    |   movel([0.140704, -1.403542, -2.555417, -0.753429, 1.570796, 1.711500],accel_mss,speed_ms,0,blend_radius_m)
    |   movel([0.140545, -1.403137, -2.555717, -0.753535, 1.570796, 1.711342],accel_mss,speed_ms,0,blend_radius_m)
    |   movel([0.140518, -1.402670, -2.556062, -0.753657, 1.570796, 1.711315],accel_mss,speed_ms,0,blend_radius_m)
    |   movel([0.140843, -1.401367, -2.557021, -0.754000, 1.570796, 1.711640],accel_mss,speed_ms,0,blend_radius_m)
    |   movel([0.141778, -1.399330, -2.558517, -0.754541, 1.570796, 1.712574],accel_mss,speed_ms,0,blend_radius_m)
    |   movel([0.143948, -1.395292, -2.561465, -0.755632, 1.570796, 1.714744],accel_mss,speed_ms,0,blend_radius_m)
    |   movel([0.146129, -1.391761, -2.564023, -0.756605, 1.570796, 1.716925],accel_mss,speed_ms,0,blend_radius_m)
    |   movel([0.148288, -1.388770, -2.566175, -0.757443, 1.570796, 1.719084],accel_mss,speed_ms,0,blend_radius_m)
    |   movel([0.149299, -1.387556, -2.567045, -0.757787, 1.570796, 1.720095],accel_mss,speed_ms,0,blend_radius_m)
    |   movel([0.150400, -1.386385, -2.567883, -0.758121, 1.570796, 1.721196],accel_mss,speed_ms,0,blend_radius_m)
    |   movel([0.151006, -1.385809, -2.568294, -0.758286, 1.570796, 1.721802],accel_mss,speed_ms,0,blend_radius_m)
    |   movel([0.153931, -1.383309, -2.570072, -0.759008, 1.570796, 1.724727],accel_mss,speed_ms,0,blend_radius_m)
    |   movel([0.156335, -1.381241, -2.571537, -0.759611, 1.570796, 1.727131],accel_mss,speed_ms,0,blend_radius_m)
    |   movel([0.159846, -1.377963, -2.573845, -0.760581, 1.570796, 1.730642],accel_mss,speed_ms,0,blend_radius_m)
    |   movel([0.163498, -1.374419, -2.576324, -0.761646, 1.570796, 1.734295],accel_mss,speed_ms,0,blend_radius_m)
    |   movel([0.166495, -1.371353, -2.578454, -0.762582, 1.570796, 1.737291],accel_mss,speed_ms,0,blend_radius_m)
    |   movel([0.170128, -1.367386, -2.581189, -0.763813, 1.570796, 1.740924],accel_mss,speed_ms,0,blend_radius_m)
    |   movel([0.173632, -1.363310, -2.583978, -0.765102, 1.570796, 1.744429],accel_mss,speed_ms,0,blend_radius_m)
    |   movel([0.176951, -1.359183, -2.586776, -0.766430, 1.570796, 1.747747],accel_mss,speed_ms,0,blend_radius_m)
    |   movel([0.180116, -1.354961, -2.589615, -0.767813, 1.570796, 1.750913],accel_mss,speed_ms,0,blend_radius_m)
    |   movel([0.183146, -1.350616, -2.592510, -0.769263, 1.570796, 1.753942],accel_mss,speed_ms,0,blend_radius_m)
    |   movel([0.186004, -1.346192, -2.595432, -0.770766, 1.570796, 1.756800],accel_mss,speed_ms,0,blend_radius_m)
    |   movel([0.188766, -1.341570, -2.598454, -0.772364, 1.570796, 1.759562],accel_mss,speed_ms,0,blend_radius_m)
    |   movel([0.191358, -1.336888, -2.601487, -0.774014, 1.570796, 1.762154],accel_mss,speed_ms,0,blend_radius_m)
    |   movel([0.194463, -1.330702, -2.605447, -0.776239, 1.570796, 1.765259],accel_mss,speed_ms,0,blend_radius_m)
    |   movel([0.197247, -1.324446, -2.609400, -0.778543, 1.570796, 1.768044],accel_mss,speed_ms,0,blend_radius_m)
    |   movel([0.199689, -1.318160, -2.613319, -0.780910, 1.570796, 1.770485],accel_mss,speed_ms,0,blend_radius_m)
    |   movel([0.201775, -1.311845, -2.617204, -0.783340, 1.570796, 1.772572],accel_mss,speed_ms,0,blend_radius_m)
    |   movel([0.203479, -1.305580, -2.621005, -0.785804, 1.570796, 1.774275],accel_mss,speed_ms,0,blend_radius_m)
    |   movel([0.204799, -1.299337, -2.624742, -0.788310, 1.570796, 1.775595],accel_mss,speed_ms,0,blend_radius_m)
    |   movel([0.205703, -1.293227, -2.628351, -0.790810, 1.570796, 1.776499],accel_mss,speed_ms,0,blend_radius_m)
    |   movel([0.206187, -1.287198, -2.631865, -0.793325, 1.570796, 1.776984],accel_mss,speed_ms,0,blend_radius_m)
    |   movel([0.206497, -1.284112, -2.633647, -0.794631, 1.570796, 1.777293],accel_mss,speed_ms,0,blend_radius_m)
    |   movel([0.207150, -1.281572, -2.635103, -0.795714, 1.570796, 1.777946],accel_mss,speed_ms,0,blend_radius_m)
    |   movel([0.207592, -1.280512, -2.635709, -0.796168, 1.570796, 1.778388],accel_mss,speed_ms,0,blend_radius_m)
    |   movel([0.208169, -1.279450, -2.636314, -0.796625, 1.570796, 1.778966],accel_mss,speed_ms,0,blend_radius_m)
    |   movel([0.208820, -1.278512, -2.636847, -0.797030, 1.570796, 1.779616],accel_mss,speed_ms,0,blend_radius_m)
    |   movel([0.210185, -1.277059, -2.637671, -0.797659, 1.570796, 1.780981],accel_mss,speed_ms,0,blend_radius_m)
    |   movel([0.210558, -1.276782, -2.637828, -0.797779, 1.570796, 1.781354],accel_mss,speed_ms,0,blend_radius_m)
    |   movel([0.211690, -1.276412, -2.638038, -0.797940, 1.570796, 1.782486],accel_mss,speed_ms,0,blend_radius_m)
    |   movel([0.212752, -1.276292, -2.638105, -0.797992, 1.570796, 1.783548],accel_mss,speed_ms,0,blend_radius_m)
    |   movel([0.213684, -1.276450, -2.638016, -0.797923, 1.570796, 1.784480],accel_mss,speed_ms,0,blend_radius_m)
    |   movel([0.214653, -1.276937, -2.637741, -0.797712, 1.570796, 1.785449],accel_mss,speed_ms,0,blend_radius_m)
    |   movel([0.215875, -1.277874, -2.637209, -0.797305, 1.570796, 1.786671],accel_mss,speed_ms,0,blend_radius_m)
    |   movel([0.217446, -1.279458, -2.636309, -0.796622, 1.570796, 1.788242],accel_mss,speed_ms,0,blend_radius_m)
    |   movel([0.218701, -1.281264, -2.635279, -0.795846, 1.570796, 1.789497],accel_mss,speed_ms,0,blend_radius_m)
    |   movel([0.219663, -1.283334, -2.634093, -0.794961, 1.570796, 1.790460],accel_mss,speed_ms,0,blend_radius_m)
    |   movel([0.220360, -1.285698, -2.632733, -0.793959, 1.570796, 1.791157],accel_mss,speed_ms,0,blend_radius_m)
    |   movel([0.220698, -1.287639, -2.631610, -0.793140, 1.570796, 1.791494],accel_mss,speed_ms,0,blend_radius_m)
    |   movel([0.220907, -1.289828, -2.630338, -0.792223, 1.570796, 1.791703],accel_mss,speed_ms,0,blend_radius_m)
    |   movel([0.221010, -1.292587, -2.628727, -0.791076, 1.570796, 1.791806],accel_mss,speed_ms,0,blend_radius_m)
    |   movel([0.221047, -1.301875, -2.623229, -0.787285, 1.570796, 1.791843],accel_mss,speed_ms,0,blend_radius_m)
    |   movel([0.221214, -1.305714, -2.620925, -0.785751, 1.570796, 1.792010],accel_mss,speed_ms,0,blend_radius_m)
    |   movel([0.221547, -1.308582, -2.619190, -0.784617, 1.570796, 1.792343],accel_mss,speed_ms,0,blend_radius_m)
    |   movel([0.222085, -1.310928, -2.617763, -0.783698, 1.570796, 1.792881],accel_mss,speed_ms,0,blend_radius_m)
    |   movel([0.223013, -1.312969, -2.616516, -0.782904, 1.570796, 1.793809],accel_mss,speed_ms,0,blend_radius_m)
    |   movel([0.223526, -1.313486, -2.616199, -0.782704, 1.570796, 1.794322],accel_mss,speed_ms,0,blend_radius_m)
    |   movel([0.224254, -1.313767, -2.616027, -0.782595, 1.570796, 1.795050],accel_mss,speed_ms,0,blend_radius_m)
    |   movel([0.225101, -1.313780, -2.616019, -0.782590, 1.570796, 1.795897],accel_mss,speed_ms,0,blend_radius_m)
    |   movel([0.226034, -1.313522, -2.616177, -0.782690, 1.570796, 1.796830],accel_mss,speed_ms,0,blend_radius_m)
    |   movel([0.227364, -1.312916, -2.616548, -0.782924, 1.570796, 1.798160],accel_mss,speed_ms,0,blend_radius_m)
    |   movel([0.228675, -1.312190, -2.616993, -0.783206, 1.570796, 1.799471],accel_mss,speed_ms,0,blend_radius_m)
    |   movel([0.230649, -1.310918, -2.617770, -0.783702, 1.570796, 1.801445],accel_mss,speed_ms,0,blend_radius_m)
    |   movel([0.232595, -1.309499, -2.618633, -0.784257, 1.570796, 1.803392],accel_mss,speed_ms,0,blend_radius_m)
    |   movel([0.234895, -1.307655, -2.619752, -0.784982, 1.570796, 1.805692],accel_mss,speed_ms,0,blend_radius_m)
    |   movel([0.241204, -1.302298, -2.622976, -0.787115, 1.570796, 1.812000],accel_mss,speed_ms,0,blend_radius_m)
    |   movel([0.243555, -1.300425, -2.624095, -0.787869, 1.570796, 1.814351],accel_mss,speed_ms,0,blend_radius_m)
    |   movel([0.245404, -1.299103, -2.624882, -0.788405, 1.570796, 1.816201],accel_mss,speed_ms,0,blend_radius_m)
    |   movel([0.246945, -1.298199, -2.625419, -0.788772, 1.570796, 1.817741],accel_mss,speed_ms,0,blend_radius_m)
    |   movel([0.247792, -1.297825, -2.625640, -0.788924, 1.570796, 1.818588],accel_mss,speed_ms,0,blend_radius_m)
    |   movel([0.248634, -1.297559, -2.625797, -0.789032, 1.570796, 1.819430],accel_mss,speed_ms,0,blend_radius_m)
    |   movel([0.249248, -1.297496, -2.625835, -0.789058, 1.570796, 1.820044],accel_mss,speed_ms,0,blend_radius_m)
    |   movel([0.249761, -1.297629, -2.625756, -0.789004, 1.570796, 1.820557],accel_mss,speed_ms,0,blend_radius_m)
    |   movel([0.250158, -1.297955, -2.625563, -0.788871, 1.570796, 1.820954],accel_mss,speed_ms,0,blend_radius_m)
    |   movel([0.250380, -1.298428, -2.625282, -0.788679, 1.570796, 1.821176],accel_mss,speed_ms,0,blend_radius_m)
    |   movel([0.250519, -1.300019, -2.624337, -0.788033, 1.570796, 1.821316],accel_mss,speed_ms,0,blend_radius_m)
    |   movel([0.250460, -1.300588, -2.623997, -0.787803, 1.570796, 1.821256],accel_mss,speed_ms,0,blend_radius_m)
    |   movel([0.250051, -1.302510, -2.622849, -0.787030, 1.570796, 1.820848],accel_mss,speed_ms,0,blend_radius_m)
    |   speed_ms = 0.005
    |   movel([0.250051, -1.293311, -2.618501, -0.800577, 1.570796, 1.820848],accel_mss,speed_ms,0,blend_radius_m)
    |   speed_ms = 0.040
    |   movel([0.285051, -1.248291, -2.643835, -0.820263, 1.570796, 1.855847],accel_mss,speed_ms,0,blend_radius_m)
    |   speed_ms = 0.005
    |   movel([0.285051, -1.257727, -2.648387, -0.806275, 1.570796, 1.855847],accel_mss,speed_ms,0,blend_radius_m)
    |   speed_ms = 0.025
    |   movel([0.285376, -1.257416, -2.648555, -0.806417, 1.570796, 1.856173],accel_mss,speed_ms,0,blend_radius_m)
    |   movel([0.285614, -1.256958, -2.648804, -0.806628, 1.570796, 1.856410],accel_mss,speed_ms,0,blend_radius_m)
    |   movel([0.285837, -1.256166, -2.649232, -0.806991, 1.570796, 1.856634],accel_mss,speed_ms,0,blend_radius_m)
    |   movel([0.286186, -1.254460, -2.650153, -0.807777, 1.570796, 1.856982],accel_mss,speed_ms,0,blend_radius_m)
    |   movel([0.286743, -1.250478, -2.652287, -0.809624, 1.570796, 1.857539],accel_mss,speed_ms,0,blend_radius_m)
    |   movel([0.286878, -1.248468, -2.653357, -0.810563, 1.570796, 1.857674],accel_mss,speed_ms,0,blend_radius_m)
    |   movel([0.286872, -1.244744, -2.655328, -0.812317, 1.570796, 1.857668],accel_mss,speed_ms,0,blend_radius_m)
    |   movel([0.286986, -1.244540, -2.655435, -0.812414, 1.570796, 1.857783],accel_mss,speed_ms,0,blend_radius_m)
    |   movel([0.287202, -1.244420, -2.655498, -0.812470, 1.570796, 1.857998],accel_mss,speed_ms,0,blend_radius_m)
    |   movel([0.287547, -1.244241, -2.655593, -0.812555, 1.570796, 1.858343],accel_mss,speed_ms,0,blend_radius_m)
    |   movel([0.287781, -1.243914, -2.655765, -0.812710, 1.570796, 1.858577],accel_mss,speed_ms,0,blend_radius_m)
    |   movel([0.288488, -1.241734, -2.656909, -0.813747, 1.570796, 1.859284],accel_mss,speed_ms,0,blend_radius_m)
    |   movel([0.289030, -1.239404, -2.658125, -0.814861, 1.570796, 1.859827],accel_mss,speed_ms,0,blend_radius_m)
    |   movel([0.289144, -1.237626, -2.659048, -0.815715, 1.570796, 1.859940],accel_mss,speed_ms,0,blend_radius_m)
    |   movel([0.289053, -1.236830, -2.659460, -0.816098, 1.570796, 1.859850],accel_mss,speed_ms,0,blend_radius_m)
    |   movel([0.288864, -1.236454, -2.659655, -0.816280, 1.570796, 1.859660],accel_mss,speed_ms,0,blend_radius_m)
    |   movel([0.288563, -1.236423, -2.659671, -0.816295, 1.570796, 1.859359],accel_mss,speed_ms,0,blend_radius_m)
    |   movel([0.288157, -1.236673, -2.659542, -0.816174, 1.570796, 1.858953],accel_mss,speed_ms,0,blend_radius_m)
    |   movel([0.287954, -1.236902, -2.659423, -0.816064, 1.570796, 1.858750],accel_mss,speed_ms,0,blend_radius_m)
    |   movel([0.287849, -1.237125, -2.659308, -0.815956, 1.570796, 1.858646],accel_mss,speed_ms,0,blend_radius_m)
    |   movel([0.287893, -1.238385, -2.658654, -0.815350, 1.570796, 1.858690],accel_mss,speed_ms,0,blend_radius_m)
    |   movel([0.287887, -1.238901, -2.658386, -0.815102, 1.570796, 1.858683],accel_mss,speed_ms,0,blend_radius_m)
    |   movel([0.287513, -1.241756, -2.656897, -0.813736, 1.570796, 1.858309],accel_mss,speed_ms,0,blend_radius_m)
    |   movel([0.286745, -1.241225, -2.657175, -0.813990, 1.570796, 1.857541],accel_mss,speed_ms,0,blend_radius_m)
    |   movel([0.285897, -1.240581, -2.657511, -0.814297, 1.570796, 1.856693],accel_mss,speed_ms,0,blend_radius_m)
    |   movel([0.285614, -1.240567, -2.657518, -0.814304, 1.570796, 1.856410],accel_mss,speed_ms,0,blend_radius_m)
    |   movel([0.285291, -1.240759, -2.657418, -0.814212, 1.570796, 1.856087],accel_mss,speed_ms,0,blend_radius_m)
    |   movel([0.285032, -1.241098, -2.657241, -0.814050, 1.570796, 1.855828],accel_mss,speed_ms,0,blend_radius_m)
    |   movel([0.284949, -1.241441, -2.657062, -0.813886, 1.570796, 1.855745],accel_mss,speed_ms,0,blend_radius_m)
    |   movel([0.285127, -1.242733, -2.656385, -0.813271, 1.570796, 1.855923],accel_mss,speed_ms,0,blend_radius_m)
    |   movel([0.285518, -1.245087, -2.655147, -0.812155, 1.570796, 1.856314],accel_mss,speed_ms,0,blend_radius_m)
    |   movel([0.285650, -1.247822, -2.653700, -0.810866, 1.570796, 1.856446],accel_mss,speed_ms,0,blend_radius_m)
    |   movel([0.285532, -1.250774, -2.652129, -0.809486, 1.570796, 1.856328],accel_mss,speed_ms,0,blend_radius_m)
    |   movel([0.285165, -1.253795, -2.650510, -0.808083, 1.570796, 1.855962],accel_mss,speed_ms,0,blend_radius_m)
    |   movel([0.285029, -1.254644, -2.650053, -0.807692, 1.570796, 1.855825],accel_mss,speed_ms,0,blend_radius_m)
    |   movel([0.284302, -1.253909, -2.650449, -0.808031, 1.570796, 1.855098],accel_mss,speed_ms,0,blend_radius_m)
    |   movel([0.283800, -1.253480, -2.650679, -0.808229, 1.570796, 1.854597],accel_mss,speed_ms,0,blend_radius_m)
    |   movel([0.283333, -1.253283, -2.650785, -0.808320, 1.570796, 1.854130],accel_mss,speed_ms,0,blend_radius_m)
    |   movel([0.282930, -1.253309, -2.650771, -0.808308, 1.570796, 1.853726],accel_mss,speed_ms,0,blend_radius_m)
    |   movel([0.282597, -1.253538, -2.650648, -0.808202, 1.570796, 1.853393],accel_mss,speed_ms,0,blend_radius_m)
    |   movel([0.282529, -1.253687, -2.650569, -0.808134, 1.570796, 1.853326],accel_mss,speed_ms,0,blend_radius_m)
    |   movel([0.282510, -1.258156, -2.648154, -0.806079, 1.570796, 1.853306],accel_mss,speed_ms,0,blend_radius_m)
    |   movel([0.282198, -1.261061, -2.646572, -0.804757, 1.570796, 1.852994],accel_mss,speed_ms,0,blend_radius_m)
    |   movel([0.281587, -1.264059, -2.644927, -0.803402, 1.570796, 1.852383],accel_mss,speed_ms,0,blend_radius_m)
    |   movel([0.280691, -1.267080, -2.643260, -0.802049, 1.570796, 1.851487],accel_mss,speed_ms,0,blend_radius_m)
    |   movel([0.279427, -1.270591, -2.641308, -0.800490, 1.570796, 1.850224],accel_mss,speed_ms,0,blend_radius_m)
    |   movel([0.278962, -1.271746, -2.640662, -0.799981, 1.570796, 1.849758],accel_mss,speed_ms,0,blend_radius_m)
    |   movel([0.278807, -1.271873, -2.640591, -0.799925, 1.570796, 1.849604],accel_mss,speed_ms,0,blend_radius_m)
    |   movel([0.277931, -1.270373, -2.641430, -0.800587, 1.570796, 1.848727],accel_mss,speed_ms,0,blend_radius_m)
    |   movel([0.277769, -1.270303, -2.641468, -0.800618, 1.570796, 1.848565],accel_mss,speed_ms,0,blend_radius_m)
    |   movel([0.277540, -1.270378, -2.641427, -0.800584, 1.570796, 1.848337],accel_mss,speed_ms,0,blend_radius_m)
    |   movel([0.277044, -1.270862, -2.641156, -0.800370, 1.570796, 1.847840],accel_mss,speed_ms,0,blend_radius_m)
    |   movel([0.276091, -1.272411, -2.640290, -0.799688, 1.570796, 1.846887],accel_mss,speed_ms,0,blend_radius_m)
    |   movel([0.274985, -1.274185, -2.639293, -0.798910, 1.570796, 1.845782],accel_mss,speed_ms,0,blend_radius_m)
    |   movel([0.272593, -1.277484, -2.637431, -0.797474, 1.570796, 1.843389],accel_mss,speed_ms,0,blend_radius_m)
    |   movel([0.271336, -1.278966, -2.636589, -0.796834, 1.570796, 1.842132],accel_mss,speed_ms,0,blend_radius_m)
    |   movel([0.268622, -1.281745, -2.635004, -0.795640, 1.570796, 1.839418],accel_mss,speed_ms,0,blend_radius_m)
    |   movel([0.267067, -1.283243, -2.634146, -0.795001, 1.570796, 1.837863],accel_mss,speed_ms,0,blend_radius_m)
    |   movel([0.266749, -1.283416, -2.634046, -0.794927, 1.570796, 1.837545],accel_mss,speed_ms,0,blend_radius_m)
    |   movel([0.267003, -1.282685, -2.634466, -0.795238, 1.570796, 1.837799],accel_mss,speed_ms,0,blend_radius_m)
    |   movel([0.267156, -1.282373, -2.634645, -0.795372, 1.570796, 1.837953],accel_mss,speed_ms,0,blend_radius_m)
    |   movel([0.267374, -1.281632, -2.635069, -0.795688, 1.570796, 1.838171],accel_mss,speed_ms,0,blend_radius_m)
    |   movel([0.267265, -1.281398, -2.635202, -0.795788, 1.570796, 1.838061],accel_mss,speed_ms,0,blend_radius_m)
    |   movel([0.267029, -1.281290, -2.635264, -0.795835, 1.570796, 1.837826],accel_mss,speed_ms,0,blend_radius_m)
    |   movel([0.266711, -1.281327, -2.635243, -0.795819, 1.570796, 1.837507],accel_mss,speed_ms,0,blend_radius_m)
    |   movel([0.266379, -1.281504, -2.635142, -0.795743, 1.570796, 1.837175],accel_mss,speed_ms,0,blend_radius_m)
    |   movel([0.264753, -1.282545, -2.634546, -0.795298, 1.570796, 1.835550],accel_mss,speed_ms,0,blend_radius_m)
    |   movel([0.262799, -1.283498, -2.633999, -0.794892, 1.570796, 1.833595],accel_mss,speed_ms,0,blend_radius_m)
    |   movel([0.260794, -1.284240, -2.633572, -0.794576, 1.570796, 1.831590],accel_mss,speed_ms,0,blend_radius_m)
    |   movel([0.259009, -1.284664, -2.633329, -0.794397, 1.570796, 1.829805],accel_mss,speed_ms,0,blend_radius_m)
    |   movel([0.257566, -1.284887, -2.633200, -0.794302, 1.570796, 1.828363],accel_mss,speed_ms,0,blend_radius_m)
    |   movel([0.258580, -1.284223, -2.633582, -0.794583, 1.570796, 1.829377],accel_mss,speed_ms,0,blend_radius_m)
    |   movel([0.260055, -1.283172, -2.634187, -0.795031, 1.570796, 1.830851],accel_mss,speed_ms,0,blend_radius_m)
    |   movel([0.260356, -1.282858, -2.634366, -0.795164, 1.570796, 1.831153],accel_mss,speed_ms,0,blend_radius_m)
    |   movel([0.260526, -1.282508, -2.634567, -0.795314, 1.570796, 1.831322],accel_mss,speed_ms,0,blend_radius_m)
    |   movel([0.260492, -1.282266, -2.634706, -0.795417, 1.570796, 1.831289],accel_mss,speed_ms,0,blend_radius_m)
    |   movel([0.260273, -1.282178, -2.634756, -0.795455, 1.570796, 1.831070],accel_mss,speed_ms,0,blend_radius_m)
    |   movel([0.257760, -1.282555, -2.634540, -0.795294, 1.570796, 1.828556],accel_mss,speed_ms,0,blend_radius_m)
    |   movel([0.257143, -1.282548, -2.634544, -0.795297, 1.570796, 1.827940],accel_mss,speed_ms,0,blend_radius_m)
    |   movel([0.255004, -1.282200, -2.634744, -0.795445, 1.570796, 1.825800],accel_mss,speed_ms,0,blend_radius_m)
    |   movel([0.253443, -1.281754, -2.634999, -0.795636, 1.570796, 1.824239],accel_mss,speed_ms,0,blend_radius_m)
    |   movel([0.250378, -1.280508, -2.635711, -0.796170, 1.570796, 1.821175],accel_mss,speed_ms,0,blend_radius_m)
    |   movel([0.248859, -1.279752, -2.636142, -0.796495, 1.570796, 1.819656],accel_mss,speed_ms,0,blend_radius_m)
    |   movel([0.250690, -1.278643, -2.636773, -0.796973, 1.570796, 1.821486],accel_mss,speed_ms,0,blend_radius_m)
    |   movel([0.251682, -1.278031, -2.637120, -0.797238, 1.570796, 1.822478],accel_mss,speed_ms,0,blend_radius_m)
    |   movel([0.252495, -1.277367, -2.637497, -0.797525, 1.570796, 1.823292],accel_mss,speed_ms,0,blend_radius_m)
    |   movel([0.252645, -1.277082, -2.637658, -0.797649, 1.570796, 1.823441],accel_mss,speed_ms,0,blend_radius_m)
    |   movel([0.252625, -1.276826, -2.637803, -0.797760, 1.570796, 1.823422],accel_mss,speed_ms,0,blend_radius_m)
    |   movel([0.252420, -1.276660, -2.637897, -0.797832, 1.570796, 1.823216],accel_mss,speed_ms,0,blend_radius_m)
    |   movel([0.250730, -1.276368, -2.638062, -0.797959, 1.570796, 1.821526],accel_mss,speed_ms,0,blend_radius_m)
    |   movel([0.248210, -1.275930, -2.638310, -0.798149, 1.570796, 1.819007],accel_mss,speed_ms,0,blend_radius_m)
    |   movel([0.245957, -1.275281, -2.638676, -0.798432, 1.570796, 1.816753],accel_mss,speed_ms,0,blend_radius_m)
    |   movel([0.243901, -1.274399, -2.639173, -0.798817, 1.570796, 1.814697],accel_mss,speed_ms,0,blend_radius_m)
    |   movel([0.241981, -1.273254, -2.639817, -0.799318, 1.570796, 1.812778],accel_mss,speed_ms,0,blend_radius_m)
    |   movel([0.240628, -1.272326, -2.640337, -0.799726, 1.570796, 1.811424],accel_mss,speed_ms,0,blend_radius_m)
    |   movel([0.242149, -1.271884, -2.640585, -0.799920, 1.570796, 1.812945],accel_mss,speed_ms,0,blend_radius_m)
    |   movel([0.243577, -1.271407, -2.640852, -0.800130, 1.570796, 1.814374],accel_mss,speed_ms,0,blend_radius_m)
    |   movel([0.244768, -1.270870, -2.641152, -0.800367, 1.570796, 1.815564],accel_mss,speed_ms,0,blend_radius_m)
    |   movel([0.245620, -1.270334, -2.641451, -0.800604, 1.570796, 1.816416],accel_mss,speed_ms,0,blend_radius_m)
    |   movel([0.245834, -1.270117, -2.641572, -0.800700, 1.570796, 1.816631],accel_mss,speed_ms,0,blend_radius_m)
    |   movel([0.245956, -1.269872, -2.641709, -0.800808, 1.570796, 1.816753],accel_mss,speed_ms,0,blend_radius_m)
    |   movel([0.245937, -1.269634, -2.641841, -0.800913, 1.570796, 1.816733],accel_mss,speed_ms,0,blend_radius_m)
    |   movel([0.245749, -1.269477, -2.641929, -0.800983, 1.570796, 1.816546],accel_mss,speed_ms,0,blend_radius_m)
    |   movel([0.244338, -1.269231, -2.642066, -0.801092, 1.570796, 1.815134],accel_mss,speed_ms,0,blend_radius_m)
    |   movel([0.243592, -1.269121, -2.642127, -0.801141, 1.570796, 1.814389],accel_mss,speed_ms,0,blend_radius_m)
    |   movel([0.241491, -1.268600, -2.642417, -0.801372, 1.570796, 1.812287],accel_mss,speed_ms,0,blend_radius_m)
    |   movel([0.240267, -1.268026, -2.642736, -0.801628, 1.570796, 1.811064],accel_mss,speed_ms,0,blend_radius_m)
    |   movel([0.237751, -1.266229, -2.643731, -0.802429, 1.570796, 1.808548],accel_mss,speed_ms,0,blend_radius_m)
    |   movel([0.236809, -1.265256, -2.644268, -0.802865, 1.570796, 1.807606],accel_mss,speed_ms,0,blend_radius_m)
    |   movel([0.234505, -1.262022, -2.646046, -0.804321, 1.570796, 1.805301],accel_mss,speed_ms,0,blend_radius_m)
    |   movel([0.233410, -1.260262, -2.647008, -0.805119, 1.570796, 1.804207],accel_mss,speed_ms,0,blend_radius_m)
    |   movel([0.233543, -1.260074, -2.647110, -0.805205, 1.570796, 1.804339],accel_mss,speed_ms,0,blend_radius_m)
    |   movel([0.234795, -1.260230, -2.647025, -0.805134, 1.570796, 1.805592],accel_mss,speed_ms,0,blend_radius_m)
    |   movel([0.235308, -1.260299, -2.646987, -0.805102, 1.570796, 1.806104],accel_mss,speed_ms,0,blend_radius_m)
    |   movel([0.237799, -1.260349, -2.646961, -0.805080, 1.570796, 1.808596],accel_mss,speed_ms,0,blend_radius_m)
    |   movel([0.238169, -1.260286, -2.646995, -0.805108, 1.570796, 1.808965],accel_mss,speed_ms,0,blend_radius_m)
    |   movel([0.238709, -1.259961, -2.647172, -0.805256, 1.570796, 1.809505],accel_mss,speed_ms,0,blend_radius_m)
    |   movel([0.238960, -1.259624, -2.647356, -0.805410, 1.570796, 1.809756],accel_mss,speed_ms,0,blend_radius_m)
    |   movel([0.238957, -1.259371, -2.647493, -0.805524, 1.570796, 1.809753],accel_mss,speed_ms,0,blend_radius_m)
    |   movel([0.238642, -1.259153, -2.647612, -0.805624, 1.570796, 1.809439],accel_mss,speed_ms,0,blend_radius_m)
    |   movel([0.236421, -1.258302, -2.648074, -0.806012, 1.570796, 1.807218],accel_mss,speed_ms,0,blend_radius_m)
    |   movel([0.235003, -1.257497, -2.648511, -0.806380, 1.570796, 1.805800],accel_mss,speed_ms,0,blend_radius_m)
    |   movel([0.233648, -1.256526, -2.649037, -0.806826, 1.570796, 1.804444],accel_mss,speed_ms,0,blend_radius_m)
    |   movel([0.232494, -1.255470, -2.649608, -0.807311, 1.570796, 1.803290],accel_mss,speed_ms,0,blend_radius_m)
    |   movel([0.230105, -1.252420, -2.651248, -0.808720, 1.570796, 1.800901],accel_mss,speed_ms,0,blend_radius_m)
    |   movel([0.228663, -1.250377, -2.652341, -0.809671, 1.570796, 1.799459],accel_mss,speed_ms,0,blend_radius_m)
    |   movel([0.228616, -1.250017, -2.652533, -0.809839, 1.570796, 1.799412],accel_mss,speed_ms,0,blend_radius_m)
    |   movel([0.229564, -1.250008, -2.652538, -0.809843, 1.570796, 1.800360],accel_mss,speed_ms,0,blend_radius_m)
    |   movel([0.229992, -1.250043, -2.652519, -0.809827, 1.570796, 1.800788],accel_mss,speed_ms,0,blend_radius_m)
    |   movel([0.231557, -1.249933, -2.652578, -0.809878, 1.570796, 1.802353],accel_mss,speed_ms,0,blend_radius_m)
    |   movel([0.232180, -1.249807, -2.652645, -0.809937, 1.570796, 1.802977],accel_mss,speed_ms,0,blend_radius_m)
    |   movel([0.232659, -1.249546, -2.652784, -0.810059, 1.570796, 1.803455],accel_mss,speed_ms,0,blend_radius_m)
    |   movel([0.232791, -1.249316, -2.652907, -0.810167, 1.570796, 1.803588],accel_mss,speed_ms,0,blend_radius_m)
    |   movel([0.232794, -1.249067, -2.653039, -0.810283, 1.570796, 1.803590],accel_mss,speed_ms,0,blend_radius_m)
    |   movel([0.232586, -1.248795, -2.653184, -0.810410, 1.570796, 1.803382],accel_mss,speed_ms,0,blend_radius_m)
    |   movel([0.231381, -1.247999, -2.653607, -0.810783, 1.570796, 1.802178],accel_mss,speed_ms,0,blend_radius_m)
    |   movel([0.229753, -1.246883, -2.654198, -0.811308, 1.570796, 1.800549],accel_mss,speed_ms,0,blend_radius_m)
    |   movel([0.227669, -1.245075, -2.655153, -0.812160, 1.570796, 1.798465],accel_mss,speed_ms,0,blend_radius_m)
    |   movel([0.225697, -1.243153, -2.656165, -0.813072, 1.570796, 1.796493],accel_mss,speed_ms,0,blend_radius_m)
    |   movel([0.224468, -1.241636, -2.656959, -0.813793, 1.570796, 1.795264],accel_mss,speed_ms,0,blend_radius_m)
    |   movel([0.224133, -1.241124, -2.657228, -0.814038, 1.570796, 1.794929],accel_mss,speed_ms,0,blend_radius_m)
    |   movel([0.223619, -1.240166, -2.657728, -0.814496, 1.570796, 1.794415],accel_mss,speed_ms,0,blend_radius_m)
    |   movel([0.226300, -1.239267, -2.658196, -0.814926, 1.570796, 1.797097],accel_mss,speed_ms,0,blend_radius_m)
    |   movel([0.226990, -1.238984, -2.658343, -0.815062, 1.570796, 1.797786],accel_mss,speed_ms,0,blend_radius_m)
    |   movel([0.227360, -1.238690, -2.658496, -0.815203, 1.570796, 1.798157],accel_mss,speed_ms,0,blend_radius_m)
    |   movel([0.227525, -1.238345, -2.658675, -0.815369, 1.570796, 1.798322],accel_mss,speed_ms,0,blend_radius_m)
    |   movel([0.227501, -1.238151, -2.658776, -0.815462, 1.570796, 1.798297],accel_mss,speed_ms,0,blend_radius_m)
    |   movel([0.227391, -1.238029, -2.658839, -0.815521, 1.570796, 1.798188],accel_mss,speed_ms,0,blend_radius_m)
    |   movel([0.225593, -1.237852, -2.658931, -0.815606, 1.570796, 1.796390],accel_mss,speed_ms,0,blend_radius_m)
    |   movel([0.223952, -1.237328, -2.659202, -0.815858, 1.570796, 1.794749],accel_mss,speed_ms,0,blend_radius_m)
    |   movel([0.218123, -1.234687, -2.660567, -0.817135, 1.570796, 1.788919],accel_mss,speed_ms,0,blend_radius_m)
    |   movel([0.216800, -1.234048, -2.660896, -0.817445, 1.570796, 1.787597],accel_mss,speed_ms,0,blend_radius_m)
    |   movel([0.220608, -1.232835, -2.661519, -0.818035, 1.570796, 1.791404],accel_mss,speed_ms,0,blend_radius_m)
    |   movel([0.220926, -1.232640, -2.661619, -0.818130, 1.570796, 1.791722],accel_mss,speed_ms,0,blend_radius_m)
    |   movel([0.221103, -1.232409, -2.661737, -0.818243, 1.570796, 1.791900],accel_mss,speed_ms,0,blend_radius_m)
    |   movel([0.221168, -1.232051, -2.661920, -0.818417, 1.570796, 1.791964],accel_mss,speed_ms,0,blend_radius_m)
    |   movel([0.221038, -1.231793, -2.662052, -0.818543, 1.570796, 1.791834],accel_mss,speed_ms,0,blend_radius_m)
    |   movel([0.220136, -1.231236, -2.662337, -0.818816, 1.570796, 1.790932],accel_mss,speed_ms,0,blend_radius_m)
    |   movel([0.218436, -1.230663, -2.662630, -0.819096, 1.570796, 1.789232],accel_mss,speed_ms,0,blend_radius_m)
    |   movel([0.215494, -1.229992, -2.662972, -0.819425, 1.570796, 1.786290],accel_mss,speed_ms,0,blend_radius_m)
    |   movel([0.211124, -1.229342, -2.663303, -0.819744, 1.570796, 1.781921],accel_mss,speed_ms,0,blend_radius_m)
    |   movel([0.209198, -1.229270, -2.663340, -0.819780, 1.570796, 1.779994],accel_mss,speed_ms,0,blend_radius_m)
    |   movel([0.207322, -1.229351, -2.663298, -0.819740, 1.570796, 1.778118],accel_mss,speed_ms,0,blend_radius_m)
    |   movel([0.205959, -1.229442, -2.663252, -0.819695, 1.570796, 1.776755],accel_mss,speed_ms,0,blend_radius_m)
    |   movel([0.205889, -1.229255, -2.663347, -0.819787, 1.570796, 1.776685],accel_mss,speed_ms,0,blend_radius_m)
    |   movel([0.206212, -1.228981, -2.663486, -0.819921, 1.570796, 1.777008],accel_mss,speed_ms,0,blend_radius_m)
    |   movel([0.207881, -1.228399, -2.663782, -0.820207, 1.570796, 1.778677],accel_mss,speed_ms,0,blend_radius_m)
    |   movel([0.208910, -1.228042, -2.663964, -0.820384, 1.570796, 1.779707],accel_mss,speed_ms,0,blend_radius_m)
    |   movel([0.209651, -1.227627, -2.664174, -0.820588, 1.570796, 1.780447],accel_mss,speed_ms,0,blend_radius_m)
    |   movel([0.209813, -1.227371, -2.664304, -0.820714, 1.570796, 1.780610],accel_mss,speed_ms,0,blend_radius_m)
    |   movel([0.209810, -1.227135, -2.664423, -0.820831, 1.570796, 1.780606],accel_mss,speed_ms,0,blend_radius_m)
    |   movel([0.209627, -1.226934, -2.664525, -0.820930, 1.570796, 1.780424],accel_mss,speed_ms,0,blend_radius_m)
    |   movel([0.208422, -1.226483, -2.664753, -0.821153, 1.570796, 1.779219],accel_mss,speed_ms,0,blend_radius_m)
    |   movel([0.205590, -1.225749, -2.665124, -0.821516, 1.570796, 1.776387],accel_mss,speed_ms,0,blend_radius_m)
    |   movel([0.202937, -1.225278, -2.665361, -0.821749, 1.570796, 1.773733],accel_mss,speed_ms,0,blend_radius_m)
    |   movel([0.200496, -1.225073, -2.665465, -0.821852, 1.570796, 1.771292],accel_mss,speed_ms,0,blend_radius_m)
    |   movel([0.198313, -1.225138, -2.665432, -0.821819, 1.570796, 1.769109],accel_mss,speed_ms,0,blend_radius_m)
    |   movel([0.196815, -1.225270, -2.665365, -0.821754, 1.570796, 1.767612],accel_mss,speed_ms,0,blend_radius_m)
    |   movel([0.196665, -1.225161, -2.665420, -0.821808, 1.570796, 1.767461],accel_mss,speed_ms,0,blend_radius_m)
    |   movel([0.196789, -1.224942, -2.665530, -0.821916, 1.570796, 1.767585],accel_mss,speed_ms,0,blend_radius_m)
    |   movel([0.198166, -1.223979, -2.666015, -0.822395, 1.570796, 1.768963],accel_mss,speed_ms,0,blend_radius_m)
    |   movel([0.198894, -1.223467, -2.666272, -0.822649, 1.570796, 1.769690],accel_mss,speed_ms,0,blend_radius_m)
    |   movel([0.200219, -1.222435, -2.666790, -0.823164, 1.570796, 1.771015],accel_mss,speed_ms,0,blend_radius_m)
    |   movel([0.200325, -1.222080, -2.666968, -0.823342, 1.570796, 1.771122],accel_mss,speed_ms,0,blend_radius_m)
    |   movel([0.200128, -1.221809, -2.667103, -0.823477, 1.570796, 1.770925],accel_mss,speed_ms,0,blend_radius_m)
    |   movel([0.199567, -1.221632, -2.667191, -0.823565, 1.570796, 1.770363],accel_mss,speed_ms,0,blend_radius_m)
    |   movel([0.198593, -1.221552, -2.667232, -0.823605, 1.570796, 1.769390],accel_mss,speed_ms,0,blend_radius_m)
    |   movel([0.196633, -1.221578, -2.667219, -0.823592, 1.570796, 1.767430],accel_mss,speed_ms,0,blend_radius_m)
    |   movel([0.194680, -1.221799, -2.667108, -0.823482, 1.570796, 1.765476],accel_mss,speed_ms,0,blend_radius_m)
    |   movel([0.192596, -1.222232, -2.666892, -0.823266, 1.570796, 1.763392],accel_mss,speed_ms,0,blend_radius_m)
    |   movel([0.187306, -1.223836, -2.666087, -0.822466, 1.570796, 1.758102],accel_mss,speed_ms,0,blend_radius_m)
    |   movel([0.188189, -1.223147, -2.666433, -0.822809, 1.570796, 1.758986],accel_mss,speed_ms,0,blend_radius_m)
    |   movel([0.190951, -1.221398, -2.667309, -0.823682, 1.570796, 1.761748],accel_mss,speed_ms,0,blend_radius_m)
    |   movel([0.191998, -1.220793, -2.667611, -0.823985, 1.570796, 1.762794],accel_mss,speed_ms,0,blend_radius_m)
    |   movel([0.192752, -1.220193, -2.667910, -0.824286, 1.570796, 1.763549],accel_mss,speed_ms,0,blend_radius_m)
    |   movel([0.192853, -1.219933, -2.668039, -0.824416, 1.570796, 1.763650],accel_mss,speed_ms,0,blend_radius_m)
    |   movel([0.192799, -1.219732, -2.668139, -0.824517, 1.570796, 1.763595],accel_mss,speed_ms,0,blend_radius_m)
    |   movel([0.192621, -1.219642, -2.668184, -0.824563, 1.570796, 1.763417],accel_mss,speed_ms,0,blend_radius_m)
    |   movel([0.191818, -1.219665, -2.668173, -0.824551, 1.570796, 1.762614],accel_mss,speed_ms,0,blend_radius_m)
    |   movel([0.190436, -1.219979, -2.668017, -0.824394, 1.570796, 1.761232],accel_mss,speed_ms,0,blend_radius_m)
    |   movel([0.188230, -1.220663, -2.667676, -0.824051, 1.570796, 1.759026],accel_mss,speed_ms,0,blend_radius_m)
    |   movel([0.185617, -1.221590, -2.667213, -0.823586, 1.570796, 1.756413],accel_mss,speed_ms,0,blend_radius_m)
    |   movel([0.183271, -1.222559, -2.666728, -0.823102, 1.570796, 1.754068],accel_mss,speed_ms,0,blend_radius_m)
    |   movel([0.181012, -1.223650, -2.666181, -0.822559, 1.570796, 1.751808],accel_mss,speed_ms,0,blend_radius_m)
    |   movel([0.177669, -1.225509, -2.665245, -0.821635, 1.570796, 1.748465],accel_mss,speed_ms,0,blend_radius_m)
    |   movel([0.176813, -1.225982, -2.665006, -0.821401, 1.570796, 1.747609],accel_mss,speed_ms,0,blend_radius_m)
    |   movel([0.175997, -1.226380, -2.664805, -0.821204, 1.570796, 1.746794],accel_mss,speed_ms,0,blend_radius_m)
    |   movel([0.178601, -1.223460, -2.666276, -0.822653, 1.570796, 1.749397],accel_mss,speed_ms,0,blend_radius_m)
    |   movel([0.178734, -1.223160, -2.666426, -0.822803, 1.570796, 1.749531],accel_mss,speed_ms,0,blend_radius_m)
    |   movel([0.178636, -1.222956, -2.666529, -0.822904, 1.570796, 1.749432],accel_mss,speed_ms,0,blend_radius_m)
    |   movel([0.178308, -1.222902, -2.666556, -0.822931, 1.570796, 1.749105],accel_mss,speed_ms,0,blend_radius_m)
    |   movel([0.177911, -1.223021, -2.666496, -0.822872, 1.570796, 1.748708],accel_mss,speed_ms,0,blend_radius_m)
    |   movel([0.175884, -1.224088, -2.665960, -0.822340, 1.570796, 1.746681],accel_mss,speed_ms,0,blend_radius_m)
    |   movel([0.172834, -1.226022, -2.664986, -0.821381, 1.570796, 1.743630],accel_mss,speed_ms,0,blend_radius_m)
    |   movel([0.169896, -1.228324, -2.663820, -0.820245, 1.570796, 1.740693],accel_mss,speed_ms,0,blend_radius_m)
    |   movel([0.167285, -1.230813, -2.662554, -0.819023, 1.570796, 1.738081],accel_mss,speed_ms,0,blend_radius_m)
    |   movel([0.166198, -1.232033, -2.661930, -0.818427, 1.570796, 1.736995],accel_mss,speed_ms,0,blend_radius_m)
    |   movel([0.164772, -1.233885, -2.660979, -0.817524, 1.570796, 1.735569],accel_mss,speed_ms,0,blend_radius_m)
    |   movel([0.164564, -1.234101, -2.660869, -0.817420, 1.570796, 1.735360],accel_mss,speed_ms,0,blend_radius_m)
    |   movel([0.164315, -1.234041, -2.660899, -0.817449, 1.570796, 1.735111],accel_mss,speed_ms,0,blend_radius_m)
    |   movel([0.164271, -1.233832, -2.661006, -0.817550, 1.570796, 1.735067],accel_mss,speed_ms,0,blend_radius_m)
    |   movel([0.164651, -1.230126, -2.662903, -0.819359, 1.570796, 1.735447],accel_mss,speed_ms,0,blend_radius_m)
    |   movel([0.164669, -1.229441, -2.663253, -0.819695, 1.570796, 1.735465],accel_mss,speed_ms,0,blend_radius_m)
    |   movel([0.164533, -1.229162, -2.663395, -0.819832, 1.570796, 1.735329],accel_mss,speed_ms,0,blend_radius_m)
    |   movel([0.164233, -1.229131, -2.663410, -0.819848, 1.570796, 1.735029],accel_mss,speed_ms,0,blend_radius_m)
    |   movel([0.163603, -1.229470, -2.663238, -0.819681, 1.570796, 1.734399],accel_mss,speed_ms,0,blend_radius_m)
    |   movel([0.162386, -1.230459, -2.662734, -0.819196, 1.570796, 1.733182],accel_mss,speed_ms,0,blend_radius_m)
    |   movel([0.159613, -1.233064, -2.661401, -0.817924, 1.570796, 1.730409],accel_mss,speed_ms,0,blend_radius_m)
    |   movel([0.158106, -1.234701, -2.660560, -0.817128, 1.570796, 1.728902],accel_mss,speed_ms,0,blend_radius_m)
    |   movel([0.156782, -1.236322, -2.659723, -0.816344, 1.570796, 1.727578],accel_mss,speed_ms,0,blend_radius_m)
    |   movel([0.155567, -1.238024, -2.658842, -0.815524, 1.570796, 1.726364],accel_mss,speed_ms,0,blend_radius_m)
    |   movel([0.154384, -1.239908, -2.657862, -0.814619, 1.570796, 1.725180],accel_mss,speed_ms,0,blend_radius_m)
    |   movel([0.153051, -1.242162, -2.656684, -0.813543, 1.570796, 1.723847],accel_mss,speed_ms,0,blend_radius_m)
    |   movel([0.152725, -1.241096, -2.657242, -0.814051, 1.570796, 1.723521],accel_mss,speed_ms,0,blend_radius_m)
    |   movel([0.152704, -1.240568, -2.657518, -0.814303, 1.570796, 1.723500],accel_mss,speed_ms,0,blend_radius_m)
    |   movel([0.153039, -1.237608, -2.659058, -0.815724, 1.570796, 1.723836],accel_mss,speed_ms,0,blend_radius_m)
    |   movel([0.153018, -1.237264, -2.659235, -0.815889, 1.570796, 1.723815],accel_mss,speed_ms,0,blend_radius_m)
    |   movel([0.152912, -1.237181, -2.659279, -0.815929, 1.570796, 1.723708],accel_mss,speed_ms,0,blend_radius_m)
    |   movel([0.152498, -1.237285, -2.659225, -0.815879, 1.570796, 1.723294],accel_mss,speed_ms,0,blend_radius_m)
    |   movel([0.152090, -1.237574, -2.659075, -0.815740, 1.570796, 1.722886],accel_mss,speed_ms,0,blend_radius_m)
    |   movel([0.149321, -1.240339, -2.657637, -0.814413, 1.570796, 1.720118],accel_mss,speed_ms,0,blend_radius_m)
    |   movel([0.146721, -1.243098, -2.656194, -0.813098, 1.570796, 1.717518],accel_mss,speed_ms,0,blend_radius_m)
    |   movel([0.146069, -1.243894, -2.655775, -0.812720, 1.570796, 1.716865],accel_mss,speed_ms,0,blend_radius_m)
    |   movel([0.144999, -1.245485, -2.654937, -0.811967, 1.570796, 1.715796],accel_mss,speed_ms,0,blend_radius_m)
    |   movel([0.144671, -1.245405, -2.654979, -0.812005, 1.570796, 1.715467],accel_mss,speed_ms,0,blend_radius_m)
    |   movel([0.144500, -1.245218, -2.655078, -0.812093, 1.570796, 1.715296],accel_mss,speed_ms,0,blend_radius_m)
    |   movel([0.143782, -1.244501, -2.655456, -0.812432, 1.570796, 1.714579],accel_mss,speed_ms,0,blend_radius_m)
    |   movel([0.143257, -1.244905, -2.655243, -0.812241, 1.570796, 1.714054],accel_mss,speed_ms,0,blend_radius_m)
    |   movel([0.142533, -1.246161, -2.654580, -0.811648, 1.570796, 1.713330],accel_mss,speed_ms,0,blend_radius_m)
    |   movel([0.141054, -1.249263, -2.652935, -0.810191, 1.570796, 1.711851],accel_mss,speed_ms,0,blend_radius_m)
    |   movel([0.140572, -1.250503, -2.652274, -0.809612, 1.570796, 1.711369],accel_mss,speed_ms,0,blend_radius_m)
    |   movel([0.140026, -1.252586, -2.651160, -0.808644, 1.570796, 1.710822],accel_mss,speed_ms,0,blend_radius_m)
    |   movel([0.139729, -1.254358, -2.650207, -0.807823, 1.570796, 1.710525],accel_mss,speed_ms,0,blend_radius_m)
    |   movel([0.139259, -1.258283, -2.648085, -0.806021, 1.570796, 1.710055],accel_mss,speed_ms,0,blend_radius_m)
    |   movel([0.139264, -1.259179, -2.647598, -0.805612, 1.570796, 1.710061],accel_mss,speed_ms,0,blend_radius_m)
    |   movel([0.138644, -1.258541, -2.647945, -0.805903, 1.570796, 1.709440],accel_mss,speed_ms,0,blend_radius_m)
    |   movel([0.138392, -1.258138, -2.648164, -0.806087, 1.570796, 1.709189],accel_mss,speed_ms,0,blend_radius_m)
    |   movel([0.137202, -1.255731, -2.649467, -0.807191, 1.570796, 1.707998],accel_mss,speed_ms,0,blend_radius_m)
    |   movel([0.137010, -1.255613, -2.649531, -0.807245, 1.570796, 1.707806],accel_mss,speed_ms,0,blend_radius_m)
    |   movel([0.136430, -1.255734, -2.649466, -0.807190, 1.570796, 1.707227],accel_mss,speed_ms,0,blend_radius_m)
    |   movel([0.136222, -1.255949, -2.649350, -0.807091, 1.570796, 1.707018],accel_mss,speed_ms,0,blend_radius_m)
    |   movel([0.136016, -1.256389, -2.649111, -0.806888, 1.570796, 1.706812],accel_mss,speed_ms,0,blend_radius_m)
    |   movel([0.135548, -1.257659, -2.648424, -0.806307, 1.570796, 1.706345],accel_mss,speed_ms,0,blend_radius_m)
    |   movel([0.135037, -1.259523, -2.647410, -0.805455, 1.570796, 1.705833],accel_mss,speed_ms,0,blend_radius_m)
    |   movel([0.134561, -1.262508, -2.645780, -0.804102, 1.570796, 1.705357],accel_mss,speed_ms,0,blend_radius_m)
    |   movel([0.134228, -1.265449, -2.644162, -0.802778, 1.570796, 1.705024],accel_mss,speed_ms,0,blend_radius_m)
    |   movel([0.134230, -1.267251, -2.643165, -0.801973, 1.570796, 1.705027],accel_mss,speed_ms,0,blend_radius_m)
    |   movel([0.134420, -1.268595, -2.642420, -0.801375, 1.570796, 1.705216],accel_mss,speed_ms,0,blend_radius_m)
    |   movel([0.134734, -1.270003, -2.641635, -0.800750, 1.570796, 1.705530],accel_mss,speed_ms,0,blend_radius_m)
    |   movel([0.135719, -1.272718, -2.640118, -0.799554, 1.570796, 1.706516],accel_mss,speed_ms,0,blend_radius_m)
    |   movel([0.135834, -1.273034, -2.639941, -0.799415, 1.570796, 1.706630],accel_mss,speed_ms,0,blend_radius_m)
    |   movel([0.135885, -1.273379, -2.639747, -0.799263, 1.570796, 1.706681],accel_mss,speed_ms,0,blend_radius_m)
    |   movel([0.134264, -1.273139, -2.639881, -0.799369, 1.570796, 1.705061],accel_mss,speed_ms,0,blend_radius_m)
    |   movel([0.133249, -1.272945, -2.639990, -0.799454, 1.570796, 1.704046],accel_mss,speed_ms,0,blend_radius_m)
    |   movel([0.132627, -1.272963, -2.639980, -0.799446, 1.570796, 1.703424],accel_mss,speed_ms,0,blend_radius_m)
    |   movel([0.132264, -1.273172, -2.639863, -0.799354, 1.570796, 1.703060],accel_mss,speed_ms,0,blend_radius_m)
    |   movel([0.132067, -1.273540, -2.639656, -0.799193, 1.570796, 1.702863],accel_mss,speed_ms,0,blend_radius_m)
    |   movel([0.132094, -1.274771, -2.638963, -0.798654, 1.570796, 1.702891],accel_mss,speed_ms,0,blend_radius_m)
    |   movel([0.132776, -1.277596, -2.637367, -0.797426, 1.570796, 1.703573],accel_mss,speed_ms,0,blend_radius_m)
    |   movel([0.133631, -1.280555, -2.635684, -0.796150, 1.570796, 1.704427],accel_mss,speed_ms,0,blend_radius_m)
    |   movel([0.134534, -1.283033, -2.634266, -0.795090, 1.570796, 1.705330],accel_mss,speed_ms,0,blend_radius_m)
    |   movel([0.135244, -1.284762, -2.633272, -0.794355, 1.570796, 1.706040],accel_mss,speed_ms,0,blend_radius_m)
    |   movel([0.134146, -1.285952, -2.632586, -0.793851, 1.570796, 1.704942],accel_mss,speed_ms,0,blend_radius_m)
    |   movel([0.133841, -1.286480, -2.632281, -0.793628, 1.570796, 1.704637],accel_mss,speed_ms,0,blend_radius_m)
    |   movel([0.133422, -1.287771, -2.631534, -0.793085, 1.570796, 1.704219],accel_mss,speed_ms,0,blend_radius_m)
    |   movel([0.133357, -1.289089, -2.630768, -0.792532, 1.570796, 1.704153],accel_mss,speed_ms,0,blend_radius_m)
    |   movel([0.133671, -1.290206, -2.630118, -0.792065, 1.570796, 1.704468],accel_mss,speed_ms,0,blend_radius_m)
    |   movel([0.134126, -1.290747, -2.629802, -0.791839, 1.570796, 1.704922],accel_mss,speed_ms,0,blend_radius_m)
    |   movel([0.134355, -1.290796, -2.629774, -0.791819, 1.570796, 1.705151],accel_mss,speed_ms,0,blend_radius_m)
    |   movel([0.134641, -1.290689, -2.629836, -0.791864, 1.570796, 1.705438],accel_mss,speed_ms,0,blend_radius_m)
    |   movel([0.134868, -1.290468, -2.629965, -0.791956, 1.570796, 1.705664],accel_mss,speed_ms,0,blend_radius_m)
    |   movel([0.134954, -1.290215, -2.630113, -0.792061, 1.570796, 1.705750],accel_mss,speed_ms,0,blend_radius_m)
    |   movel([0.134804, -1.289483, -2.630539, -0.792367, 1.570796, 1.705600],accel_mss,speed_ms,0,blend_radius_m)
    |   movel([0.134633, -1.288853, -2.630905, -0.792631, 1.570796, 1.705429],accel_mss,speed_ms,0,blend_radius_m)
    |   movel([0.134600, -1.288044, -2.631375, -0.792970, 1.570796, 1.705396],accel_mss,speed_ms,0,blend_radius_m)
    |   movel([0.134698, -1.287211, -2.631858, -0.793320, 1.570796, 1.705494],accel_mss,speed_ms,0,blend_radius_m)
    |   movel([0.134930, -1.286516, -2.632260, -0.793613, 1.570796, 1.705726],accel_mss,speed_ms,0,blend_radius_m)
    |   movel([0.135184, -1.286066, -2.632520, -0.793803, 1.570796, 1.705980],accel_mss,speed_ms,0,blend_radius_m)
    |   movel([0.135463, -1.285773, -2.632690, -0.793927, 1.570796, 1.706259],accel_mss,speed_ms,0,blend_radius_m)
    |   movel([0.135714, -1.285678, -2.632744, -0.793967, 1.570796, 1.706510],accel_mss,speed_ms,0,blend_radius_m)
    |   movel([0.135905, -1.285772, -2.632690, -0.793927, 1.570796, 1.706701],accel_mss,speed_ms,0,blend_radius_m)
    |   movel([0.136082, -1.285854, -2.632642, -0.793892, 1.570796, 1.706878],accel_mss,speed_ms,0,blend_radius_m)
    |   movel([0.136381, -1.285796, -2.632676, -0.793917, 1.570796, 1.707177],accel_mss,speed_ms,0,blend_radius_m)
    |   movel([0.136686, -1.285630, -2.632772, -0.793987, 1.570796, 1.707482],accel_mss,speed_ms,0,blend_radius_m)
    |   movel([0.136876, -1.285414, -2.632897, -0.794079, 1.570796, 1.707672],accel_mss,speed_ms,0,blend_radius_m)
    |   movel([0.136912, -1.285263, -2.632983, -0.794143, 1.570796, 1.707708],accel_mss,speed_ms,0,blend_radius_m)
    |   movel([0.136656, -1.284439, -2.633458, -0.794492, 1.570796, 1.707452],accel_mss,speed_ms,0,blend_radius_m)
    |   movel([0.135673, -1.282213, -2.634736, -0.795440, 1.570796, 1.706469],accel_mss,speed_ms,0,blend_radius_m)
    |   movel([0.133326, -1.274952, -2.638862, -0.798576, 1.570796, 1.704122],accel_mss,speed_ms,0,blend_radius_m)
    |   movel([0.133342, -1.274697, -2.639005, -0.798687, 1.570796, 1.704138],accel_mss,speed_ms,0,blend_radius_m)
    |   movel([0.133514, -1.274425, -2.639158, -0.798805, 1.570796, 1.704311],accel_mss,speed_ms,0,blend_radius_m)
    |   movel([0.135690, -1.274653, -2.639030, -0.798706, 1.570796, 1.706487],accel_mss,speed_ms,0,blend_radius_m)
    |   movel([0.136736, -1.274605, -2.639057, -0.798727, 1.570796, 1.707532],accel_mss,speed_ms,0,blend_radius_m)
    |   movel([0.137474, -1.274365, -2.639192, -0.798832, 1.570796, 1.708270],accel_mss,speed_ms,0,blend_radius_m)
    |   movel([0.137685, -1.274197, -2.639287, -0.798905, 1.570796, 1.708481],accel_mss,speed_ms,0,blend_radius_m)
    |   movel([0.137792, -1.273976, -2.639411, -0.799002, 1.570796, 1.708588],accel_mss,speed_ms,0,blend_radius_m)
    |   movel([0.137777, -1.273823, -2.639497, -0.799069, 1.570796, 1.708574],accel_mss,speed_ms,0,blend_radius_m)
    |   movel([0.137087, -1.272324, -2.640338, -0.799726, 1.570796, 1.707883],accel_mss,speed_ms,0,blend_radius_m)
    |   movel([0.136474, -1.270940, -2.641113, -0.800336, 1.570796, 1.707270],accel_mss,speed_ms,0,blend_radius_m)
    |   movel([0.135962, -1.269299, -2.642028, -0.801062, 1.570796, 1.706758],accel_mss,speed_ms,0,blend_radius_m)
    |   movel([0.135600, -1.267567, -2.642990, -0.801832, 1.570796, 1.706396],accel_mss,speed_ms,0,blend_radius_m)
    |   movel([0.135433, -1.265921, -2.643901, -0.802567, 1.570796, 1.706229],accel_mss,speed_ms,0,blend_radius_m)
    |   movel([0.135470, -1.264436, -2.644720, -0.803233, 1.570796, 1.706266],accel_mss,speed_ms,0,blend_radius_m)
    |   movel([0.135722, -1.262165, -2.645967, -0.804257, 1.570796, 1.706518],accel_mss,speed_ms,0,blend_radius_m)
    |   movel([0.136061, -1.259899, -2.647206, -0.805284, 1.570796, 1.706858],accel_mss,speed_ms,0,blend_radius_m)
    |   movel([0.136534, -1.258321, -2.648064, -0.806004, 1.570796, 1.707330],accel_mss,speed_ms,0,blend_radius_m)
    |   movel([0.137186, -1.258948, -2.647723, -0.805717, 1.570796, 1.707982],accel_mss,speed_ms,0,blend_radius_m)
    |   movel([0.137728, -1.259625, -2.647355, -0.805409, 1.570796, 1.708524],accel_mss,speed_ms,0,blend_radius_m)
    |   movel([0.139104, -1.260707, -2.646765, -0.804917, 1.570796, 1.709901],accel_mss,speed_ms,0,blend_radius_m)
    |   movel([0.139721, -1.260930, -2.646643, -0.804816, 1.570796, 1.710517],accel_mss,speed_ms,0,blend_radius_m)
    |   movel([0.140174, -1.260939, -2.646638, -0.804812, 1.570796, 1.710970],accel_mss,speed_ms,0,blend_radius_m)
    |   movel([0.140323, -1.260838, -2.646693, -0.804858, 1.570796, 1.711119],accel_mss,speed_ms,0,blend_radius_m)
    |   movel([0.140648, -1.260367, -2.646951, -0.805072, 1.570796, 1.711444],accel_mss,speed_ms,0,blend_radius_m)
    |   movel([0.140708, -1.260067, -2.647114, -0.805208, 1.570796, 1.711504],accel_mss,speed_ms,0,blend_radius_m)
    |   movel([0.140526, -1.258193, -2.648134, -0.806062, 1.570796, 1.711323],accel_mss,speed_ms,0,blend_radius_m)
    |   movel([0.140540, -1.257336, -2.648599, -0.806454, 1.570796, 1.711337],accel_mss,speed_ms,0,blend_radius_m)
    |   movel([0.140917, -1.254345, -2.650214, -0.807829, 1.570796, 1.711714],accel_mss,speed_ms,0,blend_radius_m)
    |   movel([0.141310, -1.252044, -2.651450, -0.808895, 1.570796, 1.712106],accel_mss,speed_ms,0,blend_radius_m)
    |   movel([0.141704, -1.250443, -2.652306, -0.809640, 1.570796, 1.712500],accel_mss,speed_ms,0,blend_radius_m)
    |   movel([0.142246, -1.248970, -2.653091, -0.810329, 1.570796, 1.713042],accel_mss,speed_ms,0,blend_radius_m)
    |   movel([0.143090, -1.247163, -2.654050, -0.811176, 1.570796, 1.713886],accel_mss,speed_ms,0,blend_radius_m)
    |   movel([0.143399, -1.246554, -2.654372, -0.811463, 1.570796, 1.714195],accel_mss,speed_ms,0,blend_radius_m)
    |   movel([0.144020, -1.246823, -2.654230, -0.811336, 1.570796, 1.714816],accel_mss,speed_ms,0,blend_radius_m)
    |   movel([0.144282, -1.246919, -2.654179, -0.811291, 1.570796, 1.715078],accel_mss,speed_ms,0,blend_radius_m)
    |   movel([0.144972, -1.246990, -2.654142, -0.811258, 1.570796, 1.715768],accel_mss,speed_ms,0,blend_radius_m)
    |   movel([0.145157, -1.246868, -2.654206, -0.811315, 1.570796, 1.715954],accel_mss,speed_ms,0,blend_radius_m)
    |   movel([0.146182, -1.245466, -2.654947, -0.811976, 1.570796, 1.716978],accel_mss,speed_ms,0,blend_radius_m)
    |   movel([0.147089, -1.244204, -2.655612, -0.812573, 1.570796, 1.717885],accel_mss,speed_ms,0,blend_radius_m)
    |   movel([0.148829, -1.242153, -2.656689, -0.813547, 1.570796, 1.719625],accel_mss,speed_ms,0,blend_radius_m)
    |   movel([0.150689, -1.240056, -2.657785, -0.814548, 1.570796, 1.721485],accel_mss,speed_ms,0,blend_radius_m)
    |   movel([0.151224, -1.239699, -2.657971, -0.814719, 1.570796, 1.722020],accel_mss,speed_ms,0,blend_radius_m)
    |   movel([0.151439, -1.240876, -2.657357, -0.814156, 1.570796, 1.722236],accel_mss,speed_ms,0,blend_radius_m)
    |   movel([0.151574, -1.241880, -2.656832, -0.813677, 1.570796, 1.722371],accel_mss,speed_ms,0,blend_radius_m)
    |   movel([0.151908, -1.242903, -2.656296, -0.813190, 1.570796, 1.722705],accel_mss,speed_ms,0,blend_radius_m)
    |   movel([0.152333, -1.243743, -2.655855, -0.812791, 1.570796, 1.723129],accel_mss,speed_ms,0,blend_radius_m)
    |   movel([0.152747, -1.244020, -2.655709, -0.812660, 1.570796, 1.723544],accel_mss,speed_ms,0,blend_radius_m)
    |   movel([0.153064, -1.243966, -2.655738, -0.812686, 1.570796, 1.723860],accel_mss,speed_ms,0,blend_radius_m)
    |   movel([0.153430, -1.243719, -2.655867, -0.812803, 1.570796, 1.724226],accel_mss,speed_ms,0,blend_radius_m)
    |   movel([0.153740, -1.243358, -2.656057, -0.812974, 1.570796, 1.724536],accel_mss,speed_ms,0,blend_radius_m)
    |   movel([0.153890, -1.242987, -2.656251, -0.813150, 1.570796, 1.724687],accel_mss,speed_ms,0,blend_radius_m)
    |   movel([0.154111, -1.242366, -2.656577, -0.813446, 1.570796, 1.724907],accel_mss,speed_ms,0,blend_radius_m)
    |   movel([0.154958, -1.240833, -2.657379, -0.814177, 1.570796, 1.725754],accel_mss,speed_ms,0,blend_radius_m)
    |   movel([0.155913, -1.239224, -2.658218, -0.814947, 1.570796, 1.726710],accel_mss,speed_ms,0,blend_radius_m)
    |   movel([0.157932, -1.236373, -2.659697, -0.816319, 1.570796, 1.728728],accel_mss,speed_ms,0,blend_radius_m)
    |   movel([0.159064, -1.235000, -2.660405, -0.816983, 1.570796, 1.729860],accel_mss,speed_ms,0,blend_radius_m)
    |   movel([0.161569, -1.232437, -2.661723, -0.818229, 1.570796, 1.732365],accel_mss,speed_ms,0,blend_radius_m)
    |   movel([0.163243, -1.230891, -2.662513, -0.818985, 1.570796, 1.734040],accel_mss,speed_ms,0,blend_radius_m)
    |   movel([0.163144, -1.231742, -2.662079, -0.818569, 1.570796, 1.733940],accel_mss,speed_ms,0,blend_radius_m)
    |   movel([0.163031, -1.233719, -2.661065, -0.817605, 1.570796, 1.733827],accel_mss,speed_ms,0,blend_radius_m)
    |   movel([0.163214, -1.235199, -2.660303, -0.816887, 1.570796, 1.734010],accel_mss,speed_ms,0,blend_radius_m)
    |   movel([0.163648, -1.236087, -2.659845, -0.816457, 1.570796, 1.734445],accel_mss,speed_ms,0,blend_radius_m)
    |   movel([0.163922, -1.236243, -2.659764, -0.816382, 1.570796, 1.734718],accel_mss,speed_ms,0,blend_radius_m)
    |   movel([0.164312, -1.236210, -2.659781, -0.816398, 1.570796, 1.735108],accel_mss,speed_ms,0,blend_radius_m)
    |   movel([0.165194, -1.234980, -2.660416, -0.816993, 1.570796, 1.735990],accel_mss,speed_ms,0,blend_radius_m)
    |   movel([0.166079, -1.233746, -2.661051, -0.817592, 1.570796, 1.736875],accel_mss,speed_ms,0,blend_radius_m)
    |   movel([0.168287, -1.231150, -2.662381, -0.818858, 1.570796, 1.739083],accel_mss,speed_ms,0,blend_radius_m)
    |   movel([0.169460, -1.229964, -2.662986, -0.819439, 1.570796, 1.740256],accel_mss,speed_ms,0,blend_radius_m)
    |   movel([0.172229, -1.227653, -2.664161, -0.820575, 1.570796, 1.743025],accel_mss,speed_ms,0,blend_radius_m)
    |   movel([0.173842, -1.226444, -2.664772, -0.821172, 1.570796, 1.744638],accel_mss,speed_ms,0,blend_radius_m)
    |   movel([0.174837, -1.225808, -2.665094, -0.821487, 1.570796, 1.745633],accel_mss,speed_ms,0,blend_radius_m)
    |   movel([0.175334, -1.225534, -2.665232, -0.821623, 1.570796, 1.746131],accel_mss,speed_ms,0,blend_radius_m)
    |   movel([0.174097, -1.227664, -2.664155, -0.820570, 1.570796, 1.744893],accel_mss,speed_ms,0,blend_radius_m)
    |   movel([0.173869, -1.228208, -2.663879, -0.820302, 1.570796, 1.744666],accel_mss,speed_ms,0,blend_radius_m)
    |   movel([0.173848, -1.228549, -2.663706, -0.820134, 1.570796, 1.744644],accel_mss,speed_ms,0,blend_radius_m)
    |   movel([0.174006, -1.228765, -2.663597, -0.820028, 1.570796, 1.744802],accel_mss,speed_ms,0,blend_radius_m)
    |   movel([0.174215, -1.228770, -2.663594, -0.820025, 1.570796, 1.745011],accel_mss,speed_ms,0,blend_radius_m)
    |   movel([0.174561, -1.228627, -2.663666, -0.820095, 1.570796, 1.745357],accel_mss,speed_ms,0,blend_radius_m)
    |   movel([0.175949, -1.227750, -2.664112, -0.820528, 1.570796, 1.746745],accel_mss,speed_ms,0,blend_radius_m)
    |   movel([0.177628, -1.226651, -2.664668, -0.821070, 1.570796, 1.748424],accel_mss,speed_ms,0,blend_radius_m)
    |   movel([0.180743, -1.224882, -2.665561, -0.821946, 1.570796, 1.751539],accel_mss,speed_ms,0,blend_radius_m)
    |   movel([0.182561, -1.223995, -2.666007, -0.822387, 1.570796, 1.753358],accel_mss,speed_ms,0,blend_radius_m)
    |   movel([0.186299, -1.222416, -2.666799, -0.823174, 1.570796, 1.757095],accel_mss,speed_ms,0,blend_radius_m)
    |   movel([0.188195, -1.221690, -2.667163, -0.823536, 1.570796, 1.758992],accel_mss,speed_ms,0,blend_radius_m)
    |   movel([0.188266, -1.221843, -2.667086, -0.823460, 1.570796, 1.759062],accel_mss,speed_ms,0,blend_radius_m)
    |   movel([0.187893, -1.222163, -2.666926, -0.823300, 1.570796, 1.758689],accel_mss,speed_ms,0,blend_radius_m)
    |   movel([0.184761, -1.224830, -2.665587, -0.821972, 1.570796, 1.755557],accel_mss,speed_ms,0,blend_radius_m)
    |   movel([0.183850, -1.225731, -2.665133, -0.821525, 1.570796, 1.754646],accel_mss,speed_ms,0,blend_radius_m)
    |   movel([0.183653, -1.226162, -2.664915, -0.821312, 1.570796, 1.754450],accel_mss,speed_ms,0,blend_radius_m)
    |   movel([0.184058, -1.226438, -2.664776, -0.821175, 1.570796, 1.754854],accel_mss,speed_ms,0,blend_radius_m)
    |   movel([0.184382, -1.226354, -2.664818, -0.821217, 1.570796, 1.755179],accel_mss,speed_ms,0,blend_radius_m)
    |   movel([0.186555, -1.225356, -2.665322, -0.821711, 1.570796, 1.757351],accel_mss,speed_ms,0,blend_radius_m)
    |   movel([0.187622, -1.224945, -2.665529, -0.821915, 1.570796, 1.758418],accel_mss,speed_ms,0,blend_radius_m)
    |   movel([0.192817, -1.223378, -2.666317, -0.822694, 1.570796, 1.763614],accel_mss,speed_ms,0,blend_radius_m)
    |   movel([0.194080, -1.223078, -2.666467, -0.822843, 1.570796, 1.764876],accel_mss,speed_ms,0,blend_radius_m)
    |   movel([0.196968, -1.222803, -2.666606, -0.822981, 1.570796, 1.767764],accel_mss,speed_ms,0,blend_radius_m)
    |   movel([0.197569, -1.222793, -2.666611, -0.822986, 1.570796, 1.768365],accel_mss,speed_ms,0,blend_radius_m)
    |   movel([0.198106, -1.222817, -2.666599, -0.822974, 1.570796, 1.768902],accel_mss,speed_ms,0,blend_radius_m)
    |   movel([0.195737, -1.224537, -2.665734, -0.822117, 1.570796, 1.766533],accel_mss,speed_ms,0,blend_radius_m)
    |   movel([0.194465, -1.225446, -2.665276, -0.821666, 1.570796, 1.765261],accel_mss,speed_ms,0,blend_radius_m)
    |   movel([0.193490, -1.226305, -2.664843, -0.821241, 1.570796, 1.764286],accel_mss,speed_ms,0,blend_radius_m)
    |   movel([0.193369, -1.226594, -2.664697, -0.821098, 1.570796, 1.764165],accel_mss,speed_ms,0,blend_radius_m)
    |   movel([0.193412, -1.226791, -2.664597, -0.821001, 1.570796, 1.764208],accel_mss,speed_ms,0,blend_radius_m)
    |   movel([0.193565, -1.226888, -2.664548, -0.820953, 1.570796, 1.764361],accel_mss,speed_ms,0,blend_radius_m)
    |   movel([0.194478, -1.226815, -2.664585, -0.820989, 1.570796, 1.765274],accel_mss,speed_ms,0,blend_radius_m)
    |   movel([0.196240, -1.226553, -2.664718, -0.821118, 1.570796, 1.767037],accel_mss,speed_ms,0,blend_radius_m)
    |   movel([0.198966, -1.226322, -2.664835, -0.821233, 1.570796, 1.769762],accel_mss,speed_ms,0,blend_radius_m)
    |   movel([0.200218, -1.226326, -2.664833, -0.821231, 1.570796, 1.771015],accel_mss,speed_ms,0,blend_radius_m)
    |   movel([0.204234, -1.226849, -2.664568, -0.820972, 1.570796, 1.775030],accel_mss,speed_ms,0,blend_radius_m)
    |   movel([0.206740, -1.227318, -2.664331, -0.820741, 1.570796, 1.777536],accel_mss,speed_ms,0,blend_radius_m)
    |   movel([0.206852, -1.227516, -2.664230, -0.820643, 1.570796, 1.777648],accel_mss,speed_ms,0,blend_radius_m)
    |   movel([0.204924, -1.228736, -2.663611, -0.820042, 1.570796, 1.775720],accel_mss,speed_ms,0,blend_radius_m)
    |   movel([0.203880, -1.229532, -2.663206, -0.819651, 1.570796, 1.774677],accel_mss,speed_ms,0,blend_radius_m)
    |   movel([0.203054, -1.230302, -2.662814, -0.819273, 1.570796, 1.773851],accel_mss,speed_ms,0,blend_radius_m)
    |   movel([0.202816, -1.230764, -2.662578, -0.819047, 1.570796, 1.773613],accel_mss,speed_ms,0,blend_radius_m)
    |   movel([0.202895, -1.230964, -2.662476, -0.818949, 1.570796, 1.773691],accel_mss,speed_ms,0,blend_radius_m)
    |   movel([0.203150, -1.231040, -2.662438, -0.818912, 1.570796, 1.773946],accel_mss,speed_ms,0,blend_radius_m)
    |   movel([0.204940, -1.230824, -2.662547, -0.819017, 1.570796, 1.775736],accel_mss,speed_ms,0,blend_radius_m)
    |   movel([0.207699, -1.230528, -2.662699, -0.819162, 1.570796, 1.778496],accel_mss,speed_ms,0,blend_radius_m)
    |   movel([0.210248, -1.230533, -2.662696, -0.819160, 1.570796, 1.781044],accel_mss,speed_ms,0,blend_radius_m)
    |   movel([0.212928, -1.230861, -2.662529, -0.818999, 1.570796, 1.783724],accel_mss,speed_ms,0,blend_radius_m)
    |   movel([0.216125, -1.231553, -2.662175, -0.818661, 1.570796, 1.786921],accel_mss,speed_ms,0,blend_radius_m)
    |   movel([0.218727, -1.232216, -2.661836, -0.818337, 1.570796, 1.789523],accel_mss,speed_ms,0,blend_radius_m)
    |   movel([0.216739, -1.232863, -2.661504, -0.818022, 1.570796, 1.787536],accel_mss,speed_ms,0,blend_radius_m)
    |   movel([0.214968, -1.233496, -2.661180, -0.817714, 1.570796, 1.785765],accel_mss,speed_ms,0,blend_radius_m)
    |   movel([0.214624, -1.233691, -2.661079, -0.817619, 1.570796, 1.785420],accel_mss,speed_ms,0,blend_radius_m)
    |   movel([0.214327, -1.233979, -2.660931, -0.817479, 1.570796, 1.785124],accel_mss,speed_ms,0,blend_radius_m)
    |   movel([0.214208, -1.234240, -2.660797, -0.817352, 1.570796, 1.785004],accel_mss,speed_ms,0,blend_radius_m)
    |   movel([0.214277, -1.234433, -2.660698, -0.817259, 1.570796, 1.785073],accel_mss,speed_ms,0,blend_radius_m)
    |   movel([0.216667, -1.235597, -2.660098, -0.816694, 1.570796, 1.787463],accel_mss,speed_ms,0,blend_radius_m)
    |   movel([0.219523, -1.236952, -2.659397, -0.816040, 1.570796, 1.790319],accel_mss,speed_ms,0,blend_radius_m)
    |   movel([0.222909, -1.238643, -2.658520, -0.815226, 1.570796, 1.793705],accel_mss,speed_ms,0,blend_radius_m)
    |   movel([0.222907, -1.238777, -2.658451, -0.815162, 1.570796, 1.793704],accel_mss,speed_ms,0,blend_radius_m)
    |   movel([0.222102, -1.239021, -2.658324, -0.815044, 1.570796, 1.792898],accel_mss,speed_ms,0,blend_radius_m)
    |   movel([0.221775, -1.239273, -2.658192, -0.814923, 1.570796, 1.792571],accel_mss,speed_ms,0,blend_radius_m)
    |   movel([0.221635, -1.239497, -2.658076, -0.814816, 1.570796, 1.792431],accel_mss,speed_ms,0,blend_radius_m)
    |   movel([0.221663, -1.239820, -2.657908, -0.814661, 1.570796, 1.792459],accel_mss,speed_ms,0,blend_radius_m)
    |   movel([0.222321, -1.240976, -2.657305, -0.814108, 1.570796, 1.793117],accel_mss,speed_ms,0,blend_radius_m)
    |   movel([0.223076, -1.242193, -2.656668, -0.813528, 1.570796, 1.793872],accel_mss,speed_ms,0,blend_radius_m)
    |   movel([0.224791, -1.244435, -2.655490, -0.812463, 1.570796, 1.795587],accel_mss,speed_ms,0,blend_radius_m)
    |   movel([0.226110, -1.245787, -2.654778, -0.811824, 1.570796, 1.796907],accel_mss,speed_ms,0,blend_radius_m)
    |   movel([0.229227, -1.248487, -2.653348, -0.810555, 1.570796, 1.800024],accel_mss,speed_ms,0,blend_radius_m)
    |   movel([0.227819, -1.247990, -2.653611, -0.810787, 1.570796, 1.798616],accel_mss,speed_ms,0,blend_radius_m)
    |   movel([0.227199, -1.247705, -2.653763, -0.810922, 1.570796, 1.797996],accel_mss,speed_ms,0,blend_radius_m)
    |   movel([0.226711, -1.247667, -2.653783, -0.810939, 1.570796, 1.797507],accel_mss,speed_ms,0,blend_radius_m)
    |   movel([0.226373, -1.247858, -2.653681, -0.810850, 1.570796, 1.797170],accel_mss,speed_ms,0,blend_radius_m)
    |   movel([0.226162, -1.248222, -2.653488, -0.810679, 1.570796, 1.796958],accel_mss,speed_ms,0,blend_radius_m)
    |   movel([0.226191, -1.248619, -2.653277, -0.810493, 1.570796, 1.796987],accel_mss,speed_ms,0,blend_radius_m)
    |   movel([0.228277, -1.252344, -2.651289, -0.808756, 1.570796, 1.799073],accel_mss,speed_ms,0,blend_radius_m)
    |   movel([0.229256, -1.253853, -2.650479, -0.808057, 1.570796, 1.800052],accel_mss,speed_ms,0,blend_radius_m)
    |   movel([0.231055, -1.256094, -2.649271, -0.807024, 1.570796, 1.801851],accel_mss,speed_ms,0,blend_radius_m)
    |   movel([0.232001, -1.257075, -2.648740, -0.806574, 1.570796, 1.802797],accel_mss,speed_ms,0,blend_radius_m)
    |   movel([0.233728, -1.258544, -2.647943, -0.805902, 1.570796, 1.804525],accel_mss,speed_ms,0,blend_radius_m)
    |   movel([0.232321, -1.258288, -2.648082, -0.806019, 1.570796, 1.803118],accel_mss,speed_ms,0,blend_radius_m)
    |   movel([0.231902, -1.258344, -2.648052, -0.805993, 1.570796, 1.802698],accel_mss,speed_ms,0,blend_radius_m)
    |   movel([0.231611, -1.258549, -2.647941, -0.805900, 1.570796, 1.802407],accel_mss,speed_ms,0,blend_radius_m)
    |   movel([0.231434, -1.258876, -2.647763, -0.805750, 1.570796, 1.802231],accel_mss,speed_ms,0,blend_radius_m)
    |   movel([0.231668, -1.259671, -2.647330, -0.805388, 1.570796, 1.802464],accel_mss,speed_ms,0,blend_radius_m)
    |   movel([0.231970, -1.260348, -2.646961, -0.805080, 1.570796, 1.802766],accel_mss,speed_ms,0,blend_radius_m)
    |   movel([0.234476, -1.264568, -2.644647, -0.803173, 1.570796, 1.805273],accel_mss,speed_ms,0,blend_radius_m)
    |   movel([0.235504, -1.265899, -2.643913, -0.802577, 1.570796, 1.806300],accel_mss,speed_ms,0,blend_radius_m)
    |   movel([0.236658, -1.267116, -2.643240, -0.802033, 1.570796, 1.807454],accel_mss,speed_ms,0,blend_radius_m)
    |   movel([0.237777, -1.268067, -2.642713, -0.801609, 1.570796, 1.808573],accel_mss,speed_ms,0,blend_radius_m)
    |   movel([0.239018, -1.268891, -2.642255, -0.801243, 1.570796, 1.809814],accel_mss,speed_ms,0,blend_radius_m)
    |   movel([0.240296, -1.269527, -2.641901, -0.800961, 1.570796, 1.811093],accel_mss,speed_ms,0,blend_radius_m)
    |   movel([0.241693, -1.270013, -2.641630, -0.800746, 1.570796, 1.812489],accel_mss,speed_ms,0,blend_radius_m)
    |   movel([0.243358, -1.270481, -2.641369, -0.800539, 1.570796, 1.814154],accel_mss,speed_ms,0,blend_radius_m)
    |   movel([0.242221, -1.270780, -2.641202, -0.800407, 1.570796, 1.813017],accel_mss,speed_ms,0,blend_radius_m)
    |   movel([0.241651, -1.270900, -2.641135, -0.800354, 1.570796, 1.812448],accel_mss,speed_ms,0,blend_radius_m)
    |   movel([0.239946, -1.270947, -2.641109, -0.800333, 1.570796, 1.810742],accel_mss,speed_ms,0,blend_radius_m)
    |   movel([0.239120, -1.270885, -2.641144, -0.800361, 1.570796, 1.809917],accel_mss,speed_ms,0,blend_radius_m)
    |   movel([0.238617, -1.270959, -2.641102, -0.800328, 1.570796, 1.809414],accel_mss,speed_ms,0,blend_radius_m)
    |   movel([0.238307, -1.271167, -2.640986, -0.800236, 1.570796, 1.809103],accel_mss,speed_ms,0,blend_radius_m)
    |   movel([0.238115, -1.271508, -2.640795, -0.800086, 1.570796, 1.808911],accel_mss,speed_ms,0,blend_radius_m)
    |   movel([0.238209, -1.271964, -2.640540, -0.799885, 1.570796, 1.809005],accel_mss,speed_ms,0,blend_radius_m)
    |   movel([0.239383, -1.273036, -2.639939, -0.799414, 1.570796, 1.810179],accel_mss,speed_ms,0,blend_radius_m)
    |   movel([0.240763, -1.274126, -2.639327, -0.798936, 1.570796, 1.811560],accel_mss,speed_ms,0,blend_radius_m)
    |   movel([0.242193, -1.275048, -2.638807, -0.798533, 1.570796, 1.812990],accel_mss,speed_ms,0,blend_radius_m)
    |   movel([0.243693, -1.275781, -2.638394, -0.798214, 1.570796, 1.814489],accel_mss,speed_ms,0,blend_radius_m)
    |   movel([0.245668, -1.276513, -2.637980, -0.797896, 1.570796, 1.816464],accel_mss,speed_ms,0,blend_radius_m)
    |   movel([0.247673, -1.277113, -2.637641, -0.797635, 1.570796, 1.818470],accel_mss,speed_ms,0,blend_radius_m)
    |   movel([0.249757, -1.277474, -2.637436, -0.797479, 1.570796, 1.820553],accel_mss,speed_ms,0,blend_radius_m)
    |   movel([0.250172, -1.277551, -2.637392, -0.797445, 1.570796, 1.820968],accel_mss,speed_ms,0,blend_radius_m)
    |   movel([0.250531, -1.277690, -2.637314, -0.797385, 1.570796, 1.821327],accel_mss,speed_ms,0,blend_radius_m)
    |   movel([0.250404, -1.277843, -2.637227, -0.797319, 1.570796, 1.821200],accel_mss,speed_ms,0,blend_radius_m)
    |   movel([0.247937, -1.279052, -2.636540, -0.796797, 1.570796, 1.818733],accel_mss,speed_ms,0,blend_radius_m)
    |   movel([0.247569, -1.279222, -2.636443, -0.796723, 1.570796, 1.818365],accel_mss,speed_ms,0,blend_radius_m)
    |   movel([0.247188, -1.279552, -2.636256, -0.796581, 1.570796, 1.817984],accel_mss,speed_ms,0,blend_radius_m)
    |   movel([0.247094, -1.279767, -2.636133, -0.796489, 1.570796, 1.817891],accel_mss,speed_ms,0,blend_radius_m)
    |   movel([0.247095, -1.280267, -2.635848, -0.796274, 1.570796, 1.817892],accel_mss,speed_ms,0,blend_radius_m)
    |   movel([0.247377, -1.280586, -2.635666, -0.796137, 1.570796, 1.818174],accel_mss,speed_ms,0,blend_radius_m)
    |   movel([0.250234, -1.281902, -2.634914, -0.795573, 1.570796, 1.821030],accel_mss,speed_ms,0,blend_radius_m)
    |   movel([0.253359, -1.283041, -2.634262, -0.795087, 1.570796, 1.824155],accel_mss,speed_ms,0,blend_radius_m)
    |   movel([0.256069, -1.283598, -2.633942, -0.794849, 1.570796, 1.826866],accel_mss,speed_ms,0,blend_radius_m)
    |   movel([0.257177, -1.283747, -2.633856, -0.794786, 1.570796, 1.827973],accel_mss,speed_ms,0,blend_radius_m)
    |   movel([0.257323, -1.283919, -2.633757, -0.794713, 1.570796, 1.828120],accel_mss,speed_ms,0,blend_radius_m)
    |   movel([0.257153, -1.284125, -2.633639, -0.794625, 1.570796, 1.827949],accel_mss,speed_ms,0,blend_radius_m)
    |   movel([0.256066, -1.284490, -2.633429, -0.794470, 1.570796, 1.826862],accel_mss,speed_ms,0,blend_radius_m)
    |   movel([0.254886, -1.284953, -2.633162, -0.794274, 1.570796, 1.825682],accel_mss,speed_ms,0,blend_radius_m)
    |   movel([0.254606, -1.285153, -2.633047, -0.794189, 1.570796, 1.825403],accel_mss,speed_ms,0,blend_radius_m)
    |   movel([0.254428, -1.285428, -2.632889, -0.794073, 1.570796, 1.825225],accel_mss,speed_ms,0,blend_radius_m)
    |   movel([0.254409, -1.285681, -2.632742, -0.793966, 1.570796, 1.825205],accel_mss,speed_ms,0,blend_radius_m)
    |   movel([0.254553, -1.285833, -2.632655, -0.793901, 1.570796, 1.825349],accel_mss,speed_ms,0,blend_radius_m)
    |   movel([0.256091, -1.286069, -2.632518, -0.793801, 1.570796, 1.826887],accel_mss,speed_ms,0,blend_radius_m)
    |   movel([0.256821, -1.286022, -2.632546, -0.793821, 1.570796, 1.827617],accel_mss,speed_ms,0,blend_radius_m)
    |   movel([0.260543, -1.285348, -2.632934, -0.794106, 1.570796, 1.831339],accel_mss,speed_ms,0,blend_radius_m)
    |   movel([0.261452, -1.285104, -2.633075, -0.794210, 1.570796, 1.832248],accel_mss,speed_ms,0,blend_radius_m)
    |   movel([0.264193, -1.283903, -2.633767, -0.794720, 1.570796, 1.834989],accel_mss,speed_ms,0,blend_radius_m)
    |   movel([0.264822, -1.283621, -2.633929, -0.794839, 1.570796, 1.835618],accel_mss,speed_ms,0,blend_radius_m)
    |   movel([0.265426, -1.283394, -2.634059, -0.794936, 1.570796, 1.836222],accel_mss,speed_ms,0,blend_radius_m)
    |   movel([0.264918, -1.284397, -2.633482, -0.794510, 1.570796, 1.835714],accel_mss,speed_ms,0,blend_radius_m)
    |   movel([0.264262, -1.285608, -2.632785, -0.793997, 1.570796, 1.835059],accel_mss,speed_ms,0,blend_radius_m)
    |   movel([0.264214, -1.285844, -2.632648, -0.793897, 1.570796, 1.835010],accel_mss,speed_ms,0,blend_radius_m)
    |   movel([0.264316, -1.286004, -2.632556, -0.793829, 1.570796, 1.835112],accel_mss,speed_ms,0,blend_radius_m)
    |   movel([0.264532, -1.286040, -2.632535, -0.793814, 1.570796, 1.835328],accel_mss,speed_ms,0,blend_radius_m)
    |   movel([0.264796, -1.285934, -2.632596, -0.793859, 1.570796, 1.835593],accel_mss,speed_ms,0,blend_radius_m)
    |   movel([0.266034, -1.285075, -2.633092, -0.794222, 1.570796, 1.836830],accel_mss,speed_ms,0,blend_radius_m)
    |   movel([0.267531, -1.283887, -2.633775, -0.794726, 1.570796, 1.838327],accel_mss,speed_ms,0,blend_radius_m)
    |   movel([0.268962, -1.282609, -2.634509, -0.795271, 1.570796, 1.839758],accel_mss,speed_ms,0,blend_radius_m)
    |   movel([0.272019, -1.279479, -2.636297, -0.796613, 1.570796, 1.842816],accel_mss,speed_ms,0,blend_radius_m)
    |   movel([0.274765, -1.276177, -2.638170, -0.798042, 1.570796, 1.845561],accel_mss,speed_ms,0,blend_radius_m)
    |   movel([0.275814, -1.274708, -2.638999, -0.798682, 1.570796, 1.846610],accel_mss,speed_ms,0,blend_radius_m)
    |   movel([0.276737, -1.273204, -2.639845, -0.799340, 1.570796, 1.847533],accel_mss,speed_ms,0,blend_radius_m)
    |   movel([0.276930, -1.272872, -2.640031, -0.799486, 1.570796, 1.847727],accel_mss,speed_ms,0,blend_radius_m)
    |   movel([0.277357, -1.272321, -2.640340, -0.799728, 1.570796, 1.848154],accel_mss,speed_ms,0,blend_radius_m)
    |   movel([0.277788, -1.273329, -2.639775, -0.799285, 1.570796, 1.848585],accel_mss,speed_ms,0,blend_radius_m)
    |   movel([0.278170, -1.274254, -2.639255, -0.798880, 1.570796, 1.848966],accel_mss,speed_ms,0,blend_radius_m)
    |   movel([0.278353, -1.274337, -2.639208, -0.798844, 1.570796, 1.849150],accel_mss,speed_ms,0,blend_radius_m)
    |   movel([0.278618, -1.274224, -2.639272, -0.798894, 1.570796, 1.849414],accel_mss,speed_ms,0,blend_radius_m)
    |   movel([0.278939, -1.273911, -2.639448, -0.799030, 1.570796, 1.849735],accel_mss,speed_ms,0,blend_radius_m)
    |   movel([0.279169, -1.273553, -2.639649, -0.799187, 1.570796, 1.849966],accel_mss,speed_ms,0,blend_radius_m)
    |   movel([0.280084, -1.271532, -2.640782, -0.800075, 1.570796, 1.850880],accel_mss,speed_ms,0,blend_radius_m)
    |   movel([0.281671, -1.267472, -2.643043, -0.801874, 1.570796, 1.852468],accel_mss,speed_ms,0,blend_radius_m)
    |   movel([0.282759, -1.263869, -2.645032, -0.803488, 1.570796, 1.853555],accel_mss,speed_ms,0,blend_radius_m)
    |   movel([0.283457, -1.260288, -2.646993, -0.805107, 1.570796, 1.854254],accel_mss,speed_ms,0,blend_radius_m)
    |   movel([0.283890, -1.256132, -2.649250, -0.807007, 1.570796, 1.854686],accel_mss,speed_ms,0,blend_radius_m)
    |   movel([0.284536, -1.257773, -2.648362, -0.806254, 1.570796, 1.855332],accel_mss,speed_ms,0,blend_radius_m)
    |   movel([0.284743, -1.257841, -2.648325, -0.806223, 1.570796, 1.855539],accel_mss,speed_ms,0,blend_radius_m)
    |   movel([0.285051, -1.257727, -2.648387, -0.806275, 1.570796, 1.855847],accel_mss,speed_ms,0,blend_radius_m)
    |   movel([0.285376, -1.257416, -2.648555, -0.806417, 1.570796, 1.856173],accel_mss,speed_ms,0,blend_radius_m)
    |   movel([0.285614, -1.256958, -2.648804, -0.806628, 1.570796, 1.856410],accel_mss,speed_ms,0,blend_radius_m)
    |   movel([0.285837, -1.256166, -2.649232, -0.806991, 1.570796, 1.856634],accel_mss,speed_ms,0,blend_radius_m)
    |   movel([0.286065, -1.255050, -2.649835, -0.807504, 1.570796, 1.856862],accel_mss,speed_ms,0,blend_radius_m)
    |   speed_ms = 0.005
    |   movel([0.286065, -1.245601, -2.645271, -0.821517, 1.570796, 1.856862],accel_mss,speed_ms,0,blend_radius_m)
    |   speed_ms = 0.040
    |   movel([0.268123, -1.229245, -2.653817, -0.829327, 1.570796, 1.838920],accel_mss,speed_ms,0,blend_radius_m)
    |   speed_ms = 0.005
    |   movel([0.268123, -1.238768, -2.658455, -0.815166, 1.570796, 1.838920],accel_mss,speed_ms,0,blend_radius_m)
    |   speed_ms = 0.025
    |   movel([0.268330, -1.240278, -2.657669, -0.814442, 1.570796, 1.839126],accel_mss,speed_ms,0,blend_radius_m)
    |   movel([0.267669, -1.239958, -2.657836, -0.814595, 1.570796, 1.838465],accel_mss,speed_ms,0,blend_radius_m)
    |   movel([0.267290, -1.239606, -2.658019, -0.814764, 1.570796, 1.838086],accel_mss,speed_ms,0,blend_radius_m)
    |   movel([0.267172, -1.239273, -2.658193, -0.814924, 1.570796, 1.837968],accel_mss,speed_ms,0,blend_radius_m)
    |   movel([0.267257, -1.238823, -2.658427, -0.815139, 1.570796, 1.838053],accel_mss,speed_ms,0,blend_radius_m)
    |   movel([0.267776, -1.237740, -2.658989, -0.815660, 1.570796, 1.838572],accel_mss,speed_ms,0,blend_radius_m)
    |   movel([0.268123, -1.238768, -2.658455, -0.815166, 1.570796, 1.838920],accel_mss,speed_ms,0,blend_radius_m)
    |   movel([0.268330, -1.240278, -2.657669, -0.814442, 1.570796, 1.839126],accel_mss,speed_ms,0,blend_radius_m)
    |   movel([0.267669, -1.239958, -2.657836, -0.814595, 1.570796, 1.838465],accel_mss,speed_ms,0,blend_radius_m)
    |   speed_ms = 0.005
    |   movel([0.267669, -1.230439, -2.653204, -0.828746, 1.570796, 1.838465],accel_mss,speed_ms,0,blend_radius_m)
    |   speed_ms = 0.040
    |   movel([0.271645, -1.189183, -2.673465, -0.849741, 1.570796, 1.842441],accel_mss,speed_ms,0,blend_radius_m)
    |   speed_ms = 0.005
    |   movel([0.271645, -1.198861, -2.678284, -0.835244, 1.570796, 1.842441],accel_mss,speed_ms,0,blend_radius_m)
    |   speed_ms = 0.025
    |   movel([0.272020, -1.198260, -2.678569, -0.835560, 1.570796, 1.842817],accel_mss,speed_ms,0,blend_radius_m)
    |   movel([0.272063, -1.197955, -2.678713, -0.835721, 1.570796, 1.842860],accel_mss,speed_ms,0,blend_radius_m)
    |   movel([0.271607, -1.197834, -2.678770, -0.835784, 1.570796, 1.842404],accel_mss,speed_ms,0,blend_radius_m)
    |   movel([0.271155, -1.197426, -2.678964, -0.835999, 1.570796, 1.841951],accel_mss,speed_ms,0,blend_radius_m)
    |   movel([0.270522, -1.196358, -2.679468, -0.836563, 1.570796, 1.841318],accel_mss,speed_ms,0,blend_radius_m)
    |   movel([0.270431, -1.195078, -2.680071, -0.837240, 1.570796, 1.841227],accel_mss,speed_ms,0,blend_radius_m)
    |   movel([0.270763, -1.193575, -2.680777, -0.838038, 1.570796, 1.841559],accel_mss,speed_ms,0,blend_radius_m)
    |   movel([0.271556, -1.191733, -2.681638, -0.839018, 1.570796, 1.842352],accel_mss,speed_ms,0,blend_radius_m)
    |   movel([0.273643, -1.188146, -2.683305, -0.840938, 1.570796, 1.844439],accel_mss,speed_ms,0,blend_radius_m)
    |   movel([0.274008, -1.187409, -2.683646, -0.841334, 1.570796, 1.844804],accel_mss,speed_ms,0,blend_radius_m)
    |   movel([0.274092, -1.186994, -2.683838, -0.841557, 1.570796, 1.844889],accel_mss,speed_ms,0,blend_radius_m)
    |   movel([0.273936, -1.186810, -2.683922, -0.841656, 1.570796, 1.844732],accel_mss,speed_ms,0,blend_radius_m)
    |   movel([0.273577, -1.186895, -2.683883, -0.841611, 1.570796, 1.844373],accel_mss,speed_ms,0,blend_radius_m)
    |   movel([0.273190, -1.187212, -2.683737, -0.841440, 1.570796, 1.843987],accel_mss,speed_ms,0,blend_radius_m)
    |   movel([0.271815, -1.189228, -2.682804, -0.840357, 1.570796, 1.842611],accel_mss,speed_ms,0,blend_radius_m)
    |   movel([0.270634, -1.191251, -2.681863, -0.839275, 1.570796, 1.841430],accel_mss,speed_ms,0,blend_radius_m)
    |   movel([0.269823, -1.192945, -2.681072, -0.838372, 1.570796, 1.840619],accel_mss,speed_ms,0,blend_radius_m)
    |   movel([0.269336, -1.194401, -2.680389, -0.837599, 1.570796, 1.840133],accel_mss,speed_ms,0,blend_radius_m)
    |   movel([0.269115, -1.196218, -2.679534, -0.836637, 1.570796, 1.839911],accel_mss,speed_ms,0,blend_radius_m)
    |   movel([0.269051, -1.196652, -2.679329, -0.836407, 1.570796, 1.839848],accel_mss,speed_ms,0,blend_radius_m)
    |   movel([0.268866, -1.197118, -2.679109, -0.836162, 1.570796, 1.839663],accel_mss,speed_ms,0,blend_radius_m)
    |   movel([0.268459, -1.197542, -2.678909, -0.835938, 1.570796, 1.839256],accel_mss,speed_ms,0,blend_radius_m)
    |   movel([0.267240, -1.199633, -2.677917, -0.834838, 1.570796, 1.838037],accel_mss,speed_ms,0,blend_radius_m)
    |   movel([0.266758, -1.200707, -2.677406, -0.834276, 1.570796, 1.837554],accel_mss,speed_ms,0,blend_radius_m)
    |   movel([0.266120, -1.202821, -2.676396, -0.833171, 1.570796, 1.836916],accel_mss,speed_ms,0,blend_radius_m)
    |   movel([0.266005, -1.203456, -2.676092, -0.832841, 1.570796, 1.836801],accel_mss,speed_ms,0,blend_radius_m)
    |   movel([0.265960, -1.205101, -2.675302, -0.831986, 1.570796, 1.836756],accel_mss,speed_ms,0,blend_radius_m)
    |   movel([0.266285, -1.206688, -2.674536, -0.831164, 1.570796, 1.837082],accel_mss,speed_ms,0,blend_radius_m)
    |   movel([0.266847, -1.207874, -2.673963, -0.830552, 1.570796, 1.837643],accel_mss,speed_ms,0,blend_radius_m)
    |   movel([0.267118, -1.208076, -2.673865, -0.830448, 1.570796, 1.837914],accel_mss,speed_ms,0,blend_radius_m)
    |   movel([0.267528, -1.208074, -2.673866, -0.830449, 1.570796, 1.838324],accel_mss,speed_ms,0,blend_radius_m)
    |   movel([0.267938, -1.207861, -2.673969, -0.830559, 1.570796, 1.838734],accel_mss,speed_ms,0,blend_radius_m)
    |   movel([0.268159, -1.207525, -2.674132, -0.830732, 1.570796, 1.838955],accel_mss,speed_ms,0,blend_radius_m)
    |   movel([0.268142, -1.207040, -2.674366, -0.830982, 1.570796, 1.838938],accel_mss,speed_ms,0,blend_radius_m)
    |   movel([0.267861, -1.206410, -2.674671, -0.831308, 1.570796, 1.838657],accel_mss,speed_ms,0,blend_radius_m)
    |   movel([0.267663, -1.205994, -2.674871, -0.831523, 1.570796, 1.838459],accel_mss,speed_ms,0,blend_radius_m)
    |   movel([0.267238, -1.204511, -2.675585, -0.832292, 1.570796, 1.838034],accel_mss,speed_ms,0,blend_radius_m)
    |   movel([0.267245, -1.203375, -2.676131, -0.832883, 1.570796, 1.838042],accel_mss,speed_ms,0,blend_radius_m)
    |   movel([0.267527, -1.201933, -2.676821, -0.833635, 1.570796, 1.838323],accel_mss,speed_ms,0,blend_radius_m)
    |   movel([0.268014, -1.200429, -2.677539, -0.834421, 1.570796, 1.838810],accel_mss,speed_ms,0,blend_radius_m)
    |   movel([0.269339, -1.197895, -2.678742, -0.835752, 1.570796, 1.840136],accel_mss,speed_ms,0,blend_radius_m)
    |   movel([0.269878, -1.198462, -2.678473, -0.835454, 1.570796, 1.840674],accel_mss,speed_ms,0,blend_radius_m)
    |   movel([0.270786, -1.199008, -2.678214, -0.835167, 1.570796, 1.841582],accel_mss,speed_ms,0,blend_radius_m)
    |   movel([0.271250, -1.199028, -2.678205, -0.835156, 1.570796, 1.842046],accel_mss,speed_ms,0,blend_radius_m)
    |   movel([0.271645, -1.198861, -2.678284, -0.835244, 1.570796, 1.842441],accel_mss,speed_ms,0,blend_radius_m)
    |   movel([0.272020, -1.198260, -2.678569, -0.835560, 1.570796, 1.842817],accel_mss,speed_ms,0,blend_radius_m)
    |   movel([0.272063, -1.197955, -2.678713, -0.835721, 1.570796, 1.842860],accel_mss,speed_ms,0,blend_radius_m)
    |   movel([0.271607, -1.197834, -2.678770, -0.835784, 1.570796, 1.842404],accel_mss,speed_ms,0,blend_radius_m)
    |   movel([0.271155, -1.197426, -2.678964, -0.835999, 1.570796, 1.841951],accel_mss,speed_ms,0,blend_radius_m)
    |   movel([0.270883, -1.196965, -2.679182, -0.836242, 1.570796, 1.841680],accel_mss,speed_ms,0,blend_radius_m)
    |   speed_ms = 0.005
    |   movel([0.270883, -1.187280, -2.674354, -0.850754, 1.570796, 1.841680],accel_mss,speed_ms,0,blend_radius_m)
    |   speed_ms = 0.040
    |   movel([0.255364, -1.189309, -2.673406, -0.849674, 1.570796, 1.826160],accel_mss,speed_ms,0,blend_radius_m)
    |   speed_ms = 0.005
    |   movel([0.255364, -1.198987, -2.678224, -0.835178, 1.570796, 1.826160],accel_mss,speed_ms,0,blend_radius_m)
    |   speed_ms = 0.025
    |   movel([0.255678, -1.198694, -2.678363, -0.835332, 1.570796, 1.826474],accel_mss,speed_ms,0,blend_radius_m)
    |   movel([0.255840, -1.198369, -2.678517, -0.835503, 1.570796, 1.826636],accel_mss,speed_ms,0,blend_radius_m)
    |   movel([0.255901, -1.197836, -2.678770, -0.835784, 1.570796, 1.826698],accel_mss,speed_ms,0,blend_radius_m)
    |   movel([0.255835, -1.192451, -2.681303, -0.838635, 1.570796, 1.826631],accel_mss,speed_ms,0,blend_radius_m)
    |   movel([0.255666, -1.191484, -2.681754, -0.839151, 1.570796, 1.826462],accel_mss,speed_ms,0,blend_radius_m)
    |   movel([0.255378, -1.190849, -2.682050, -0.839490, 1.570796, 1.826174],accel_mss,speed_ms,0,blend_radius_m)
    |   movel([0.254779, -1.190287, -2.682312, -0.839790, 1.570796, 1.825575],accel_mss,speed_ms,0,blend_radius_m)
    |   movel([0.254012, -1.190021, -2.682435, -0.839932, 1.570796, 1.824808],accel_mss,speed_ms,0,blend_radius_m)
    |   movel([0.252957, -1.190035, -2.682429, -0.839925, 1.570796, 1.823754],accel_mss,speed_ms,0,blend_radius_m)
    |   movel([0.251480, -1.190326, -2.682294, -0.839769, 1.570796, 1.822277],accel_mss,speed_ms,0,blend_radius_m)
    |   movel([0.250086, -1.190717, -2.682112, -0.839560, 1.570796, 1.820882],accel_mss,speed_ms,0,blend_radius_m)
    |   movel([0.249402, -1.191061, -2.681951, -0.839376, 1.570796, 1.820199],accel_mss,speed_ms,0,blend_radius_m)
    |   movel([0.249082, -1.191479, -2.681756, -0.839153, 1.570796, 1.819878],accel_mss,speed_ms,0,blend_radius_m)
    |   movel([0.249025, -1.192044, -2.681493, -0.838852, 1.570796, 1.819821],accel_mss,speed_ms,0,blend_radius_m)
    |   movel([0.249079, -1.192521, -2.681270, -0.838598, 1.570796, 1.819875],accel_mss,speed_ms,0,blend_radius_m)
    |   movel([0.248890, -1.192736, -2.681170, -0.838484, 1.570796, 1.819687],accel_mss,speed_ms,0,blend_radius_m)
    |   movel([0.248360, -1.192798, -2.681141, -0.838451, 1.570796, 1.819156],accel_mss,speed_ms,0,blend_radius_m)
    |   movel([0.246899, -1.193219, -2.680944, -0.838227, 1.570796, 1.817695],accel_mss,speed_ms,0,blend_radius_m)
    |   movel([0.246340, -1.193446, -2.680837, -0.838106, 1.570796, 1.817137],accel_mss,speed_ms,0,blend_radius_m)
    |   movel([0.245053, -1.194140, -2.680512, -0.837737, 1.570796, 1.815849],accel_mss,speed_ms,0,blend_radius_m)
    |   movel([0.244514, -1.194565, -2.680312, -0.837512, 1.570796, 1.815310],accel_mss,speed_ms,0,blend_radius_m)
    |   movel([0.243101, -1.196023, -2.679626, -0.836740, 1.570796, 1.813898],accel_mss,speed_ms,0,blend_radius_m)
    |   movel([0.242544, -1.196830, -2.679245, -0.836313, 1.570796, 1.813340],accel_mss,speed_ms,0,blend_radius_m)
    |   movel([0.242212, -1.197576, -2.678893, -0.835920, 1.570796, 1.813009],accel_mss,speed_ms,0,blend_radius_m)
    |   movel([0.242100, -1.198261, -2.678568, -0.835559, 1.570796, 1.812897],accel_mss,speed_ms,0,blend_radius_m)
    |   movel([0.242223, -1.198598, -2.678409, -0.835382, 1.570796, 1.813019],accel_mss,speed_ms,0,blend_radius_m)
    |   movel([0.242382, -1.198641, -2.678388, -0.835360, 1.570796, 1.813178],accel_mss,speed_ms,0,blend_radius_m)
    |   movel([0.242896, -1.198509, -2.678451, -0.835429, 1.570796, 1.813693],accel_mss,speed_ms,0,blend_radius_m)
    |   movel([0.243071, -1.198378, -2.678513, -0.835498, 1.570796, 1.813867],accel_mss,speed_ms,0,blend_radius_m)
    |   movel([0.243534, -1.197180, -2.679080, -0.836129, 1.570796, 1.814330],accel_mss,speed_ms,0,blend_radius_m)
    |   movel([0.243903, -1.196534, -2.679385, -0.836470, 1.570796, 1.814700],accel_mss,speed_ms,0,blend_radius_m)
    |   movel([0.244382, -1.195943, -2.679664, -0.836782, 1.570796, 1.815178],accel_mss,speed_ms,0,blend_radius_m)
    |   movel([0.244955, -1.195426, -2.679907, -0.837056, 1.570796, 1.815751],accel_mss,speed_ms,0,blend_radius_m)
    |   movel([0.245688, -1.194932, -2.680140, -0.837317, 1.570796, 1.816484],accel_mss,speed_ms,0,blend_radius_m)
    |   movel([0.246440, -1.194562, -2.680313, -0.837513, 1.570796, 1.817237],accel_mss,speed_ms,0,blend_radius_m)
    |   movel([0.248295, -1.193986, -2.680584, -0.837819, 1.570796, 1.819091],accel_mss,speed_ms,0,blend_radius_m)
    |   movel([0.249941, -1.193635, -2.680748, -0.838005, 1.570796, 1.820737],accel_mss,speed_ms,0,blend_radius_m)
    |   movel([0.250179, -1.192710, -2.681182, -0.838497, 1.570796, 1.820976],accel_mss,speed_ms,0,blend_radius_m)
    |   movel([0.250441, -1.192015, -2.681507, -0.838868, 1.570796, 1.821237],accel_mss,speed_ms,0,blend_radius_m)
    |   movel([0.250810, -1.191610, -2.681695, -0.839083, 1.570796, 1.821606],accel_mss,speed_ms,0,blend_radius_m)
    |   movel([0.251370, -1.191392, -2.681797, -0.839200, 1.570796, 1.822166],accel_mss,speed_ms,0,blend_radius_m)
    |   movel([0.252376, -1.191308, -2.681837, -0.839245, 1.570796, 1.823172],accel_mss,speed_ms,0,blend_radius_m)
    |   movel([0.253611, -1.191472, -2.681760, -0.839157, 1.570796, 1.824407],accel_mss,speed_ms,0,blend_radius_m)
    |   movel([0.254268, -1.192048, -2.681491, -0.838850, 1.570796, 1.825064],accel_mss,speed_ms,0,blend_radius_m)
    |   movel([0.254552, -1.193318, -2.680897, -0.838174, 1.570796, 1.825348],accel_mss,speed_ms,0,blend_radius_m)
    |   movel([0.254588, -1.197275, -2.679035, -0.836079, 1.570796, 1.825384],accel_mss,speed_ms,0,blend_radius_m)
    |   movel([0.254619, -1.198257, -2.678570, -0.835562, 1.570796, 1.825415],accel_mss,speed_ms,0,blend_radius_m)
    |   movel([0.254736, -1.199196, -2.678125, -0.835068, 1.570796, 1.825533],accel_mss,speed_ms,0,blend_radius_m)
    |   movel([0.255364, -1.198987, -2.678224, -0.835178, 1.570796, 1.826160],accel_mss,speed_ms,0,blend_radius_m)
    |   movel([0.255678, -1.198694, -2.678363, -0.835332, 1.570796, 1.826474],accel_mss,speed_ms,0,blend_radius_m)
    |   movel([0.255840, -1.198369, -2.678517, -0.835503, 1.570796, 1.826636],accel_mss,speed_ms,0,blend_radius_m)
    |   movel([0.255901, -1.197836, -2.678770, -0.835784, 1.570796, 1.826698],accel_mss,speed_ms,0,blend_radius_m)
    |   movel([0.255882, -1.196235, -2.679526, -0.836628, 1.570796, 1.826679],accel_mss,speed_ms,0,blend_radius_m)
    |   speed_ms = 0.005
    |   movel([0.255882, -1.186548, -2.674695, -0.851146, 1.570796, 1.826679],accel_mss,speed_ms,0,blend_radius_m)
    |   speed_ms = 0.040
    |   movel([0.250854, -1.179920, -2.677758, -0.854712, 1.570796, 1.821651],accel_mss,speed_ms,0,blend_radius_m)
    |   speed_ms = 0.005
    |   movel([0.250854, -1.189627, -2.682618, -0.840143, 1.570796, 1.821651],accel_mss,speed_ms,0,blend_radius_m)
    |   speed_ms = 0.025
    |   movel([0.251172, -1.189391, -2.682728, -0.840270, 1.570796, 1.821968],accel_mss,speed_ms,0,blend_radius_m)
    |   movel([0.251351, -1.189062, -2.682881, -0.840446, 1.570796, 1.822147],accel_mss,speed_ms,0,blend_radius_m)
    |   movel([0.251397, -1.188034, -2.683357, -0.840998, 1.570796, 1.822193],accel_mss,speed_ms,0,blend_radius_m)
    |   movel([0.250998, -1.186701, -2.683973, -0.841715, 1.570796, 1.821794],accel_mss,speed_ms,0,blend_radius_m)
    |   movel([0.250169, -1.185263, -2.684635, -0.842491, 1.570796, 1.820965],accel_mss,speed_ms,0,blend_radius_m)
    |   movel([0.249306, -1.184311, -2.685072, -0.843006, 1.570796, 1.820103],accel_mss,speed_ms,0,blend_radius_m)
    |   movel([0.248204, -1.183573, -2.685410, -0.843405, 1.570796, 1.819000],accel_mss,speed_ms,0,blend_radius_m)
    |   movel([0.247051, -1.183150, -2.685604, -0.843635, 1.570796, 1.817847],accel_mss,speed_ms,0,blend_radius_m)
    |   movel([0.245860, -1.183222, -2.685571, -0.843596, 1.570796, 1.816657],accel_mss,speed_ms,0,blend_radius_m)
    |   movel([0.245698, -1.183205, -2.685579, -0.843605, 1.570796, 1.816494],accel_mss,speed_ms,0,blend_radius_m)
    |   movel([0.245602, -1.183016, -2.685665, -0.843707, 1.570796, 1.816398],accel_mss,speed_ms,0,blend_radius_m)
    |   movel([0.245643, -1.182466, -2.685917, -0.844007, 1.570796, 1.816440],accel_mss,speed_ms,0,blend_radius_m)
    |   movel([0.245465, -1.182044, -2.686109, -0.844236, 1.570796, 1.816261],accel_mss,speed_ms,0,blend_radius_m)
    |   movel([0.243475, -1.179779, -2.687140, -0.845470, 1.570796, 1.814271],accel_mss,speed_ms,0,blend_radius_m)
    |   movel([0.241371, -1.177716, -2.688074, -0.846599, 1.570796, 1.812167],accel_mss,speed_ms,0,blend_radius_m)
    |   movel([0.240764, -1.177305, -2.688260, -0.846824, 1.570796, 1.811560],accel_mss,speed_ms,0,blend_radius_m)
    |   movel([0.240028, -1.177060, -2.688370, -0.846959, 1.570796, 1.810825],accel_mss,speed_ms,0,blend_radius_m)
    |   movel([0.238980, -1.177001, -2.688397, -0.846991, 1.570796, 1.809776],accel_mss,speed_ms,0,blend_radius_m)
    |   movel([0.237783, -1.177214, -2.688301, -0.846874, 1.570796, 1.808580],accel_mss,speed_ms,0,blend_radius_m)
    |   movel([0.236602, -1.177662, -2.688098, -0.846628, 1.570796, 1.807399],accel_mss,speed_ms,0,blend_radius_m)
    |   movel([0.235619, -1.178289, -2.687815, -0.846285, 1.570796, 1.806415],accel_mss,speed_ms,0,blend_radius_m)
    |   movel([0.234888, -1.178978, -2.687503, -0.845908, 1.570796, 1.805684],accel_mss,speed_ms,0,blend_radius_m)
    |   movel([0.234231, -1.179803, -2.687129, -0.845457, 1.570796, 1.805027],accel_mss,speed_ms,0,blend_radius_m)
    |   movel([0.233721, -1.180659, -2.686740, -0.844990, 1.570796, 1.804518],accel_mss,speed_ms,0,blend_radius_m)
    |   movel([0.233307, -1.181875, -2.686187, -0.844328, 1.570796, 1.804104],accel_mss,speed_ms,0,blend_radius_m)
    |   movel([0.233167, -1.182084, -2.686091, -0.844214, 1.570796, 1.803964],accel_mss,speed_ms,0,blend_radius_m)
    |   movel([0.232432, -1.182384, -2.685954, -0.844051, 1.570796, 1.803228],accel_mss,speed_ms,0,blend_radius_m)
    |   movel([0.231250, -1.182799, -2.685764, -0.843825, 1.570796, 1.802046],accel_mss,speed_ms,0,blend_radius_m)
    |   movel([0.228358, -1.184237, -2.685106, -0.843046, 1.570796, 1.799155],accel_mss,speed_ms,0,blend_radius_m)
    |   movel([0.227307, -1.184931, -2.684788, -0.842671, 1.570796, 1.798103],accel_mss,speed_ms,0,blend_radius_m)
    |   movel([0.225912, -1.186207, -2.684201, -0.841981, 1.570796, 1.796709],accel_mss,speed_ms,0,blend_radius_m)
    |   movel([0.225607, -1.186575, -2.684031, -0.841783, 1.570796, 1.796404],accel_mss,speed_ms,0,blend_radius_m)
    |   movel([0.225013, -1.187628, -2.683545, -0.841216, 1.570796, 1.795809],accel_mss,speed_ms,0,blend_radius_m)
    |   movel([0.224791, -1.188604, -2.683093, -0.840692, 1.570796, 1.795588],accel_mss,speed_ms,0,blend_radius_m)
    |   movel([0.225005, -1.189128, -2.682850, -0.840411, 1.570796, 1.795802],accel_mss,speed_ms,0,blend_radius_m)
    |   movel([0.225242, -1.189186, -2.682823, -0.840380, 1.570796, 1.796038],accel_mss,speed_ms,0,blend_radius_m)
    |   movel([0.225546, -1.189076, -2.682874, -0.840439, 1.570796, 1.796342],accel_mss,speed_ms,0,blend_radius_m)
    |   movel([0.225715, -1.188930, -2.682942, -0.840517, 1.570796, 1.796511],accel_mss,speed_ms,0,blend_radius_m)
    |   movel([0.226101, -1.188030, -2.683359, -0.841000, 1.570796, 1.796897],accel_mss,speed_ms,0,blend_radius_m)
    |   movel([0.226335, -1.187412, -2.683645, -0.841332, 1.570796, 1.797132],accel_mss,speed_ms,0,blend_radius_m)
    |   movel([0.226734, -1.186803, -2.683926, -0.841660, 1.570796, 1.797530],accel_mss,speed_ms,0,blend_radius_m)
    |   movel([0.227305, -1.186186, -2.684210, -0.841993, 1.570796, 1.798102],accel_mss,speed_ms,0,blend_radius_m)
    |   movel([0.228846, -1.185089, -2.684715, -0.842585, 1.570796, 1.799642],accel_mss,speed_ms,0,blend_radius_m)
    |   movel([0.229757, -1.184637, -2.684922, -0.842829, 1.570796, 1.800553],accel_mss,speed_ms,0,blend_radius_m)
    |   movel([0.232963, -1.183522, -2.685434, -0.843433, 1.570796, 1.803759],accel_mss,speed_ms,0,blend_radius_m)
    |   movel([0.233725, -1.183256, -2.685556, -0.843578, 1.570796, 1.804521],accel_mss,speed_ms,0,blend_radius_m)
    |   movel([0.234552, -1.182875, -2.685730, -0.843784, 1.570796, 1.805348],accel_mss,speed_ms,0,blend_radius_m)
    |   movel([0.234665, -1.182704, -2.685808, -0.843877, 1.570796, 1.805461],accel_mss,speed_ms,0,blend_radius_m)
    |   movel([0.234788, -1.181673, -2.686279, -0.844438, 1.570796, 1.805584],accel_mss,speed_ms,0,blend_radius_m)
    |   movel([0.234792, -1.181166, -2.686509, -0.844713, 1.570796, 1.805588],accel_mss,speed_ms,0,blend_radius_m)
    |   movel([0.234969, -1.180481, -2.686821, -0.845087, 1.570796, 1.805766],accel_mss,speed_ms,0,blend_radius_m)
    |   movel([0.235177, -1.180126, -2.686982, -0.845280, 1.570796, 1.805973],accel_mss,speed_ms,0,blend_radius_m)
    |   movel([0.235988, -1.179259, -2.687376, -0.845754, 1.570796, 1.806785],accel_mss,speed_ms,0,blend_radius_m)
    |   movel([0.237028, -1.178635, -2.687658, -0.846095, 1.570796, 1.807825],accel_mss,speed_ms,0,blend_radius_m)
    |   movel([0.238162, -1.178342, -2.687791, -0.846256, 1.570796, 1.808958],accel_mss,speed_ms,0,blend_radius_m)
    |   movel([0.239232, -1.178426, -2.687753, -0.846210, 1.570796, 1.810028],accel_mss,speed_ms,0,blend_radius_m)
    |   movel([0.239970, -1.178788, -2.687590, -0.846012, 1.570796, 1.810766],accel_mss,speed_ms,0,blend_radius_m)
    |   movel([0.241074, -1.179730, -2.687162, -0.845497, 1.570796, 1.811871],accel_mss,speed_ms,0,blend_radius_m)
    |   movel([0.243502, -1.182390, -2.685951, -0.844048, 1.570796, 1.814298],accel_mss,speed_ms,0,blend_radius_m)
    |   movel([0.244468, -1.183618, -2.685390, -0.843381, 1.570796, 1.815264],accel_mss,speed_ms,0,blend_radius_m)
    |   movel([0.243189, -1.184860, -2.684820, -0.842709, 1.570796, 1.813985],accel_mss,speed_ms,0,blend_radius_m)
    |   movel([0.242893, -1.185251, -2.684640, -0.842497, 1.570796, 1.813689],accel_mss,speed_ms,0,blend_radius_m)
    |   movel([0.242130, -1.186343, -2.684138, -0.841908, 1.570796, 1.812926],accel_mss,speed_ms,0,blend_radius_m)
    |   movel([0.241802, -1.186563, -2.684036, -0.841789, 1.570796, 1.812599],accel_mss,speed_ms,0,blend_radius_m)
    |   movel([0.240309, -1.187277, -2.683707, -0.841405, 1.570796, 1.811106],accel_mss,speed_ms,0,blend_radius_m)
    |   movel([0.239374, -1.187874, -2.683431, -0.841084, 1.570796, 1.810170],accel_mss,speed_ms,0,blend_radius_m)
    |   movel([0.238469, -1.188605, -2.683093, -0.840691, 1.570796, 1.809265],accel_mss,speed_ms,0,blend_radius_m)
    |   movel([0.237583, -1.189475, -2.682689, -0.840225, 1.570796, 1.808379],accel_mss,speed_ms,0,blend_radius_m)
    |   movel([0.236683, -1.190567, -2.682181, -0.839640, 1.570796, 1.807479],accel_mss,speed_ms,0,blend_radius_m)
    |   movel([0.236131, -1.191540, -2.681728, -0.839121, 1.570796, 1.806927],accel_mss,speed_ms,0,blend_radius_m)
    |   movel([0.236039, -1.192175, -2.681432, -0.838782, 1.570796, 1.806835],accel_mss,speed_ms,0,blend_radius_m)
    |   movel([0.236150, -1.192351, -2.681350, -0.838689, 1.570796, 1.806946],accel_mss,speed_ms,0,blend_radius_m)
    |   movel([0.236565, -1.192333, -2.681358, -0.838698, 1.570796, 1.807361],accel_mss,speed_ms,0,blend_radius_m)
    |   movel([0.236769, -1.192177, -2.681431, -0.838781, 1.570796, 1.807565],accel_mss,speed_ms,0,blend_radius_m)
    |   movel([0.237233, -1.191542, -2.681727, -0.839120, 1.570796, 1.808029],accel_mss,speed_ms,0,blend_radius_m)
    |   movel([0.238258, -1.190150, -2.682375, -0.839863, 1.570796, 1.809054],accel_mss,speed_ms,0,blend_radius_m)
    |   movel([0.239519, -1.188968, -2.682925, -0.840497, 1.570796, 1.810315],accel_mss,speed_ms,0,blend_radius_m)
    |   movel([0.240856, -1.188132, -2.683312, -0.840945, 1.570796, 1.811653],accel_mss,speed_ms,0,blend_radius_m)
    |   movel([0.242104, -1.187757, -2.683485, -0.841147, 1.570796, 1.812900],accel_mss,speed_ms,0,blend_radius_m)
    |   movel([0.242798, -1.187625, -2.683546, -0.841218, 1.570796, 1.813594],accel_mss,speed_ms,0,blend_radius_m)
    |   movel([0.243221, -1.187389, -2.683655, -0.841345, 1.570796, 1.814017],accel_mss,speed_ms,0,blend_radius_m)
    |   movel([0.243497, -1.187004, -2.683833, -0.841552, 1.570796, 1.814294],accel_mss,speed_ms,0,blend_radius_m)
    |   movel([0.243940, -1.185606, -2.684477, -0.842306, 1.570796, 1.814736],accel_mss,speed_ms,0,blend_radius_m)
    |   movel([0.244169, -1.185310, -2.684614, -0.842466, 1.570796, 1.814965],accel_mss,speed_ms,0,blend_radius_m)
    |   movel([0.244990, -1.184601, -2.684939, -0.842849, 1.570796, 1.815786],accel_mss,speed_ms,0,blend_radius_m)
    |   movel([0.245274, -1.184455, -2.685006, -0.842928, 1.570796, 1.816070],accel_mss,speed_ms,0,blend_radius_m)
    |   movel([0.246177, -1.184480, -2.684995, -0.842914, 1.570796, 1.816973],accel_mss,speed_ms,0,blend_radius_m)
    |   movel([0.247190, -1.184842, -2.684828, -0.842719, 1.570796, 1.817986],accel_mss,speed_ms,0,blend_radius_m)
    |   movel([0.248262, -1.185719, -2.684425, -0.842245, 1.570796, 1.819058],accel_mss,speed_ms,0,blend_radius_m)
    |   movel([0.249220, -1.186908, -2.683877, -0.841604, 1.570796, 1.820016],accel_mss,speed_ms,0,blend_radius_m)
    |   movel([0.250436, -1.189369, -2.682739, -0.840282, 1.570796, 1.821232],accel_mss,speed_ms,0,blend_radius_m)
    |   movel([0.250659, -1.189620, -2.682622, -0.840147, 1.570796, 1.821456],accel_mss,speed_ms,0,blend_radius_m)
    |   movel([0.250854, -1.189627, -2.682618, -0.840143, 1.570796, 1.821651],accel_mss,speed_ms,0,blend_radius_m)
    |   movel([0.251172, -1.189391, -2.682728, -0.840270, 1.570796, 1.821968],accel_mss,speed_ms,0,blend_radius_m)
    |   movel([0.251351, -1.189062, -2.682881, -0.840446, 1.570796, 1.822147],accel_mss,speed_ms,0,blend_radius_m)
    |   movel([0.251397, -1.188034, -2.683357, -0.840998, 1.570796, 1.822193],accel_mss,speed_ms,0,blend_radius_m)
    |   movel([0.251098, -1.187042, -2.683815, -0.841531, 1.570796, 1.821895],accel_mss,speed_ms,0,blend_radius_m)
    |   speed_ms = 0.005
    |   movel([0.251098, -1.177326, -2.678943, -0.856120, 1.570796, 1.821895],accel_mss,speed_ms,0,blend_radius_m)
    |   speed_ms = 0.040
    |   movel([0.286619, -1.175258, -2.679883, -0.857247, 1.570796, 1.857415],accel_mss,speed_ms,0,blend_radius_m)
    |   speed_ms = 0.005
    |   movel([0.286619, -1.184980, -2.684765, -0.842644, 1.570796, 1.857415],accel_mss,speed_ms,0,blend_radius_m)
    |   speed_ms = 0.025
    |   movel([0.286888, -1.184698, -2.684895, -0.842796, 1.570796, 1.857685],accel_mss,speed_ms,0,blend_radius_m)
    |   movel([0.287131, -1.184139, -2.685151, -0.843099, 1.570796, 1.857927],accel_mss,speed_ms,0,blend_radius_m)
    |   movel([0.287047, -1.183997, -2.685216, -0.843176, 1.570796, 1.857843],accel_mss,speed_ms,0,blend_radius_m)
    |   movel([0.285131, -1.183987, -2.685221, -0.843181, 1.570796, 1.855927],accel_mss,speed_ms,0,blend_radius_m)
    |   movel([0.284397, -1.183801, -2.685306, -0.843282, 1.570796, 1.855193],accel_mss,speed_ms,0,blend_radius_m)
    |   movel([0.283820, -1.183462, -2.685461, -0.843466, 1.570796, 1.854616],accel_mss,speed_ms,0,blend_radius_m)
    |   movel([0.283401, -1.182958, -2.685692, -0.843739, 1.570796, 1.854198],accel_mss,speed_ms,0,blend_radius_m)
